// TwinCAT 3 PLC project PLC
// ProgramVersion: 3.1.4023.0
// libraries:
//   Tc2_Standard, * (Beckhoff Automation GmbH)
//   Tc2_System, * (Beckhoff Automation GmbH)
//   Tc3_Module, * (Beckhoff Automation GmbH)
// project tree:
//   / PlcTask.TcTTO
//   POUs/ MAIN.TcPOU
//   DUTs/IO/PdoEntries/ Status_B0753356.TcDUT, Status_05CE4FB5.TcDUT, Status_F2CE6D91.TcDUT, Status_AE4D73AB.TcDUT, Status_D1785240.TcDUT, Ctrl_AEDC374E.TcDUT, Status_36309700.TcDUT, Control_BD9A418F.TcDUT
//   DUTs/IO/PDOs/ InfoData_6F19DB2B.TcDUT, Channel_31CEFA7F.TcDUT, WcState_9091E0EB.TcDUT, Input_Type_NC_5EE69541.TcDUT, InfoData_32EB74EA.TcDUT, Channel_42CA91F7.TcDUT, WcState_0B2B16F9.TcDUT, AI_Standard_Channel_A8DF64E3.TcDUT, Ch_1_Al_Inputs_4794C083.TcDUT, InfoData_90184F0C.TcDUT, Ch_1_A1FAE759.TcDUT, AI_Standard_Channel_4A394481.TcDUT, AI_Standard_Channel_3D09D60D.TcDUT, RMB_Status_EE6B49B4.TcDUT, RMB_Value_INT_E9189C4B.TcDUT, RMB_Control_4997AEF6.TcDUT, AO_Output_Channel_BA7EBB7C.TcDUT, Ch_1_29D41289.TcDUT, ENC_Status_compact_BFB16BB4.TcDUT, ENC_Control_compact_2ED727EF.TcDUT, Status_Us_B1E819A2.TcDUT, Status_Up_B1E819A2.TcDUT, Status_Us_In_B1E819A2.TcDUT, Status_Us_Out_B1E819A2.TcDUT, Status_Uin_449D6AB5.TcDUT, Status_Uex_449D6AB5.TcDUT, Status_Uin_627CC56E.TcDUT, Status_Uex_834F3050.TcDUT, InfoData_E68C61CD.TcDUT, InfoData_2A97D6CF.TcDUT, Inputs_25A0042B.TcDUT, Outputs_2397A10E.TcDUT
//   DUTs/IO/Boxes/ EK1100_1FC0878B.TcDUT, EK1122_1FC0878B.TcDUT, ELX1052_6CC2DB6A.TcDUT, ELX1054_EF479B4E.TcDUT, ELX1058_7670813D.TcDUT, ELX2002_B0214940.TcDUT, ELX2008_E2806B95.TcDUT, ELX3152_AA20D87B.TcDUT, ELX3158_35AE5324.TcDUT, ELX3181_05065F7B.TcDUT, ELX3202_27F12237.TcDUT, ELX3204_B6248F5B.TcDUT, ELX3252_7FD1684B.TcDUT, ELX3312_BE98AB26.TcDUT, ELX3314_E65CDB1C.TcDUT, ELX3351_DF51302B.TcDUT, ELX4154_AB92710E.TcDUT, ELX4181_0949A6C0.TcDUT, ELX5151_C163EA3C.TcDUT, ELX9410_6BC01D14.TcDUT, ELX9410_089FA854.TcDUT, ELX9560_883C11A3.TcDUT, ELX9560_F22EDCF2.TcDUT
//   DUTs/IO/Devices/ SyncUnitTask_2D604ED5.TcDUT, SyncUnitTasks_6FEB8257.TcDUT, SyncUnits_99E584AF.TcDUT
//   DUTs/IO/Topology/ Beckhoff_ELXxxxxEK1122_3FD8C7C7.TcDUT, Beckhoff_ELXxxxx_62AA317A.TcDUT, EtherCAT_Master_ELXxxxx_D0B2812D.TcDUT
//   DUTs/IO/Base/ EtcSlaveBase_82538BE2.TcDUT, EtcSlaveBase_82538BE2.TcDUT, EtcSlaveBase_82538BE2.TcDUT, EtcSlaveTerminalBase_947E5A46.TcDUT, EtcSlaveBoxBase_77A0E4A7.TcDUT, EtcSlaveEndTerminalBase_866C7F0C.TcDUT, InputBase_8311D824.TcDUT, OutputBase_10CEE7DE.TcDUT, EtcMasterBase_62654B43.TcDUT
//   GVLs/ GVL_iXlinker.TcGVL
// real-time tasks:
//   TASK PlcTask: cycle T#10ms, priority 20, ADS port 350
// I/O:
//   DEVICE EtherCAT_Master_ELXxxxx, AmsNetId 172.20.30.238.11.1
//     Beckhoff ELXxxxx [EK1100 EtherCAT Coupler (2A E-Bus)]
//       Beckhoff ELXxxxxEK1122 [EK1122 2 port EtherCAT junction]
//         Beckhoff ELXxxxxsub EK1100 [EK1100 EtherCAT Coupler (2A E-Bus)]
//       A_0001(ELX1052-0000-0016) [ELX1052 2Ch. Dig. Input  NAMUR, Ex i]
//       A_0002(ELX1054-0000-0016) [ELX1054 4Ch. Dig. Input NAMUR, NO/NC, Ex i]
//       A_0003(ELX1058-0000-0016) [ELX1058 8Ch. Dig. Input NAMUR, NO/NC, Ex i]
//       A_0004(ELX2002-0000-0016) [ELX2002 2Ch. Dig. Output 24V, 45mA, Ex i]
//       A_0005(ELX2008-0000-0016) [ELX2008 8Ch. Dig. Output 24V, 30mA, Ex i]
//       A_0006(ELX3152-0000-0016) [ELX3152 2Ch. Ana. Input 0/4-20mA, Ex i]
//       A_0007(ELX3152-0000-0017) [ELX3152 2Ch. Ana. Input 0/4-20mA, Ex i]
//       A_0008(ELX3152-0090-0016) [ELX3152-0090 2Ch. Ana. Input 0/4-20mA, Ex i, TwinSAFE SC]
//       A_0009(ELX3152-0090-0017) [ELX3152-0090 2Ch. Ana. Input 0/4-20mA, Ex i, TwinSAFE SC]
//       A_0010(ELX3158-0000-0016) [ELX3158 8Ch. Ana. Input 4-20mA, Ex i]
//       A_0011(ELX3181-0000-0016) [ELX3181 1Ch. Ana. Input 4-20mA, HART, Ex i]
//         modules: Ch. 1, Ch. 1, Ch. 1, Ch. 1, Ch. 1, Ch. 1, Ch. 1, Ch. 1
//       A_0012(ELX3181-0000-0017) [ELX3181 1Ch. Ana. Input 4-20mA, HART, Ex i]
//         modules: Ch. 1, Ch. 1, Ch. 1, Ch. 1, Ch. 1, Ch. 1, Ch. 1, Ch. 1
//       A_0013(ELX3202-0000-0016) [ELX3202 2Ch. Ana. Input PT100 (RTD), Ex i]
//       A_0014(ELX3202-0090-0016) [ELX3202-0090 2Ch. Ana. Input PT100 (RTD), Ex i, TwinSAFE SC]
//       A_0015(ELX3204-0000-0016) [ELX3204 4Ch. Ana. Input PT100 (RTD), Ex i]
//       A_0016(ELX3204-0090-0016) [ELX3204-0090 4Ch. Ana. Input PT100 (RTD), Ex i, TwinSAFE SC]
//       A_0017(ELX3252-0000-0016) [ELX3252 2Ch. Ana. Input Potentiometer measurement, Ex i]
//       A_0018(ELX3312-0000-0016) [ELX3312 2Ch. Ana Input Thermocouple (TC), Ex i]
//       A_0019(ELX3312-0090-0016) [ELX3312-0090 2Ch. Ana Input Thermocouple (TC), Ex i, TwinSAFE SC]
//       A_0020(ELX3314-0000-0016) [ELX3314 4Ch. Ana Input Thermocouple (TC), Ex i]
//       A_0021(ELX3314-0090-0016) [ELX3314-0090 4Ch. Ana Input Thermocouple (TC), Ex i, TwinSAFE SC]
//       A_0022(ELX3351-0000-0016) [ELX3351 1-channel precise load cell analysis, Ex i]
//       A_0023(ELX3351-0090-0016) [ELX3351-0090 1-channel precise load cell analysis, TwinSAFE SC, Ex i]
//       A_0024(ELX4154-0000-0016) [ELX4154 4Ch. Ana. Output 4-20mA, 16 Bit, Ex i]
//       A_0025(ELX4181-0000-0016) [ELX4181 1-channel analog output terminal 0/4...20 mA, single-ended, HART, 16 bit, Ex i]
//         modules: Ch. 1
//       A_0026(ELX4181-0000-0017) [ELX4181 1-channel analog output terminal 0/4...20 mA, single-ended, HART, 16 bit, Ex i]
//         modules: Ch. 1
//       A_0027(ELX5151-0000-0016) [ELX5151 1Ch. Inc. Encoder NAMUR, Ex i]
//       A_0028(ELX5151-0090-0016) [ELX5151-0090 1Ch. Inc. Encoder NAMUR, Ex i, TwinSAFE SC]
//       A_0030(ELX9410-0000-0016) [ELX9410 E-Bus Power Supplier (Diagnostics)]
//       A_0031(ELX9410-0000-0017) [ELX9410 E-Bus Power Supplier (Diagnostics)]
//       A_0032(ELX9410-0000-0018) [ELX9410 E-Bus Power Supplier (Diagnostics)]
//       A_0033(ELX9560-0000-0016) [ELX9560 Power supply terminal 24V DC (350mA, isolated)]
//       A_0034(ELX9560-0000-0017) [ELX9560 Power supply terminal 24V DC (650mA, isolated)]
//       A_0035(ELX9560-0000-0018) [ELX9560 Power supply terminal 24V DC (650mA, isolated)]
// variable links:
//   PLC/PLC Instance <-> EtherCAT Master ELXxxxx/Beckhoff ELXxxxx
//     PlcTask Inputs/GVL_iXlinker.EtherCAT_Master_ELXxxxx.Beckhoff_ELXxxxx.InfoData.State <-> InfoData/State
//   PLC/PLC Instance <-> EtherCAT Master ELXxxxx/Beckhoff ELXxxxx/Beckhoff ELXxxxxEK1122
//     PlcTask Inputs/GVL_iXlinker.EtherCAT_Master_ELXxxxx.Beckhoff_ELXxxxx.Beckhoff_ELXxxxxEK1122.InfoData.State <-> InfoData/State
//   PLC/PLC Instance <-> EtherCAT Master ELXxxxx/Beckhoff ELXxxxx/Beckhoff ELXxxxxEK1122/Beckhoff ELXxxxxsub EK1100
//     PlcTask Inputs/GVL_iXlinker.EtherCAT_Master_ELXxxxx.Beckhoff_ELXxxxx.Beckhoff_ELXxxxxEK1122.Beckhoff_ELXxxxxsub_EK1100.InfoData.State <-> InfoData/State
//   PLC/PLC Instance <-> EtherCAT Master ELXxxxx/Beckhoff ELXxxxx/A_0001(ELX1052-0000-0016)
//     PlcTask Inputs/GVL_iXlinker.EtherCAT_Master_ELXxxxx.Beckhoff_ELXxxxx.A_0001_ELX1052_0000_0016.Channel_1.Input <-> Channel 1/Input
//     PlcTask Inputs/GVL_iXlinker.EtherCAT_Master_ELXxxxx.Beckhoff_ELXxxxx.A_0001_ELX1052_0000_0016.Channel_2.Input <-> Channel 2/Input
//     PlcTask Inputs/GVL_iXlinker.EtherCAT_Master_ELXxxxx.Beckhoff_ELXxxxx.A_0001_ELX1052_0000_0016.Channel_1.Error <-> Channel 1/Error
//     PlcTask Inputs/GVL_iXlinker.EtherCAT_Master_ELXxxxx.Beckhoff_ELXxxxx.A_0001_ELX1052_0000_0016.Channel_2.Error <-> Channel 2/Error
//     PlcTask Inputs/GVL_iXlinker.EtherCAT_Master_ELXxxxx.Beckhoff_ELXxxxx.A_0001_ELX1052_0000_0016.WcState.WcState <-> WcState/WcState
//     PlcTask Inputs/GVL_iXlinker.EtherCAT_Master_ELXxxxx.Beckhoff_ELXxxxx.A_0001_ELX1052_0000_0016.WcState.InputToggle <-> WcState/InputToggle
//     PlcTask Inputs/GVL_iXlinker.EtherCAT_Master_ELXxxxx.Beckhoff_ELXxxxx.A_0001_ELX1052_0000_0016.InfoData.State <-> InfoData/State
//   PLC/PLC Instance <-> EtherCAT Master ELXxxxx/Beckhoff ELXxxxx/A_0002(ELX1054-0000-0016)
//     PlcTask Inputs/GVL_iXlinker.EtherCAT_Master_ELXxxxx.Beckhoff_ELXxxxx.A_0002_ELX1054_0000_0016.Channel_1.Input <-> Channel 1/Input
//     PlcTask Inputs/GVL_iXlinker.EtherCAT_Master_ELXxxxx.Beckhoff_ELXxxxx.A_0002_ELX1054_0000_0016.Channel_2.Input <-> Channel 2/Input
//     PlcTask Inputs/GVL_iXlinker.EtherCAT_Master_ELXxxxx.Beckhoff_ELXxxxx.A_0002_ELX1054_0000_0016.Channel_3.Input <-> Channel 3/Input
//     PlcTask Inputs/GVL_iXlinker.EtherCAT_Master_ELXxxxx.Beckhoff_ELXxxxx.A_0002_ELX1054_0000_0016.Channel_4.Input <-> Channel 4/Input
//     PlcTask Inputs/GVL_iXlinker.EtherCAT_Master_ELXxxxx.Beckhoff_ELXxxxx.A_0002_ELX1054_0000_0016.Channel_1.Error <-> Channel 1/Error
//     PlcTask Inputs/GVL_iXlinker.EtherCAT_Master_ELXxxxx.Beckhoff_ELXxxxx.A_0002_ELX1054_0000_0016.Channel_2.Error <-> Channel 2/Error
//     PlcTask Inputs/GVL_iXlinker.EtherCAT_Master_ELXxxxx.Beckhoff_ELXxxxx.A_0002_ELX1054_0000_0016.Channel_3.Error <-> Channel 3/Error
//     PlcTask Inputs/GVL_iXlinker.EtherCAT_Master_ELXxxxx.Beckhoff_ELXxxxx.A_0002_ELX1054_0000_0016.Channel_4.Error <-> Channel 4/Error
//     PlcTask Inputs/GVL_iXlinker.EtherCAT_Master_ELXxxxx.Beckhoff_ELXxxxx.A_0002_ELX1054_0000_0016.Input_Type_NC.Channel[0] <-> Input Type NC/Channel 1
//     PlcTask Inputs/GVL_iXlinker.EtherCAT_Master_ELXxxxx.Beckhoff_ELXxxxx.A_0002_ELX1054_0000_0016.Input_Type_NC.Channel[1] <-> Input Type NC/Channel 2
//     PlcTask Inputs/GVL_iXlinker.EtherCAT_Master_ELXxxxx.Beckhoff_ELXxxxx.A_0002_ELX1054_0000_0016.Input_Type_NC.Channel[2] <-> Input Type NC/Channel 3
//     PlcTask Inputs/GVL_iXlinker.EtherCAT_Master_ELXxxxx.Beckhoff_ELXxxxx.A_0002_ELX1054_0000_0016.Input_Type_NC.Channel[3] <-> Input Type NC/Channel 4
//     PlcTask Inputs/GVL_iXlinker.EtherCAT_Master_ELXxxxx.Beckhoff_ELXxxxx.A_0002_ELX1054_0000_0016.WcState.WcState <-> WcState/WcState
//     PlcTask Inputs/GVL_iXlinker.EtherCAT_Master_ELXxxxx.Beckhoff_ELXxxxx.A_0002_ELX1054_0000_0016.WcState.InputToggle <-> WcState/InputToggle
//     PlcTask Inputs/GVL_iXlinker.EtherCAT_Master_ELXxxxx.Beckhoff_ELXxxxx.A_0002_ELX1054_0000_0016.InfoData.State <-> InfoData/State
//   PLC/PLC Instance <-> EtherCAT Master ELXxxxx/Beckhoff ELXxxxx/A_0003(ELX1058-0000-0016)
//     PlcTask Inputs/GVL_iXlinker.EtherCAT_Master_ELXxxxx.Beckhoff_ELXxxxx.A_0003_ELX1058_0000_0016.Channel_1.Input <-> Channel 1/Input
//     PlcTask Inputs/GVL_iXlinker.EtherCAT_Master_ELXxxxx.Beckhoff_ELXxxxx.A_0003_ELX1058_0000_0016.Channel_2.Input <-> Channel 2/Input
//     PlcTask Inputs/GVL_iXlinker.EtherCAT_Master_ELXxxxx.Beckhoff_ELXxxxx.A_0003_ELX1058_0000_0016.Channel_3.Input <-> Channel 3/Input
//     PlcTask Inputs/GVL_iXlinker.EtherCAT_Master_ELXxxxx.Beckhoff_ELXxxxx.A_0003_ELX1058_0000_0016.Channel_4.Input <-> Channel 4/Input
//     PlcTask Inputs/GVL_iXlinker.EtherCAT_Master_ELXxxxx.Beckhoff_ELXxxxx.A_0003_ELX1058_0000_0016.Channel_5.Input <-> Channel 5/Input
//     PlcTask Inputs/GVL_iXlinker.EtherCAT_Master_ELXxxxx.Beckhoff_ELXxxxx.A_0003_ELX1058_0000_0016.Channel_6.Input <-> Channel 6/Input
//     PlcTask Inputs/GVL_iXlinker.EtherCAT_Master_ELXxxxx.Beckhoff_ELXxxxx.A_0003_ELX1058_0000_0016.Channel_7.Input <-> Channel 7/Input
//     PlcTask Inputs/GVL_iXlinker.EtherCAT_Master_ELXxxxx.Beckhoff_ELXxxxx.A_0003_ELX1058_0000_0016.Channel_8.Input <-> Channel 8/Input
//     PlcTask Inputs/GVL_iXlinker.EtherCAT_Master_ELXxxxx.Beckhoff_ELXxxxx.A_0003_ELX1058_0000_0016.Channel_1.Error <-> Channel 1/Error
//     PlcTask Inputs/GVL_iXlinker.EtherCAT_Master_ELXxxxx.Beckhoff_ELXxxxx.A_0003_ELX1058_0000_0016.Channel_2.Error <-> Channel 2/Error
//     PlcTask Inputs/GVL_iXlinker.EtherCAT_Master_ELXxxxx.Beckhoff_ELXxxxx.A_0003_ELX1058_0000_0016.Channel_3.Error <-> Channel 3/Error
//     PlcTask Inputs/GVL_iXlinker.EtherCAT_Master_ELXxxxx.Beckhoff_ELXxxxx.A_0003_ELX1058_0000_0016.Channel_4.Error <-> Channel 4/Error
//     PlcTask Inputs/GVL_iXlinker.EtherCAT_Master_ELXxxxx.Beckhoff_ELXxxxx.A_0003_ELX1058_0000_0016.Channel_5.Error <-> Channel 5/Error
//     PlcTask Inputs/GVL_iXlinker.EtherCAT_Master_ELXxxxx.Beckhoff_ELXxxxx.A_0003_ELX1058_0000_0016.Channel_6.Error <-> Channel 6/Error
//     PlcTask Inputs/GVL_iXlinker.EtherCAT_Master_ELXxxxx.Beckhoff_ELXxxxx.A_0003_ELX1058_0000_0016.Channel_7.Error <-> Channel 7/Error
//     PlcTask Inputs/GVL_iXlinker.EtherCAT_Master_ELXxxxx.Beckhoff_ELXxxxx.A_0003_ELX1058_0000_0016.Channel_8.Error <-> Channel 8/Error
//     PlcTask Inputs/GVL_iXlinker.EtherCAT_Master_ELXxxxx.Beckhoff_ELXxxxx.A_0003_ELX1058_0000_0016.WcState.WcState <-> WcState/WcState
//     PlcTask Inputs/GVL_iXlinker.EtherCAT_Master_ELXxxxx.Beckhoff_ELXxxxx.A_0003_ELX1058_0000_0016.WcState.InputToggle <-> WcState/InputToggle
//     PlcTask Inputs/GVL_iXlinker.EtherCAT_Master_ELXxxxx.Beckhoff_ELXxxxx.A_0003_ELX1058_0000_0016.InfoData.AdsAddr <-> InfoData/AdsAddr
//     PlcTask Inputs/GVL_iXlinker.EtherCAT_Master_ELXxxxx.Beckhoff_ELXxxxx.A_0003_ELX1058_0000_0016.InfoData.State <-> InfoData/State
//   PLC/PLC Instance <-> EtherCAT Master ELXxxxx/Beckhoff ELXxxxx/A_0004(ELX2002-0000-0016)
//     PlcTask Outputs/GVL_iXlinker.EtherCAT_Master_ELXxxxx.Beckhoff_ELXxxxx.A_0004_ELX2002_0000_0016.Channel_1.Output <-> Channel 1/Output
//     PlcTask Outputs/GVL_iXlinker.EtherCAT_Master_ELXxxxx.Beckhoff_ELXxxxx.A_0004_ELX2002_0000_0016.Channel_2.Output <-> Channel 2/Output
//     PlcTask Inputs/GVL_iXlinker.EtherCAT_Master_ELXxxxx.Beckhoff_ELXxxxx.A_0004_ELX2002_0000_0016.WcState.WcState <-> WcState/WcState
//     PlcTask Inputs/GVL_iXlinker.EtherCAT_Master_ELXxxxx.Beckhoff_ELXxxxx.A_0004_ELX2002_0000_0016.InfoData.State <-> InfoData/State
//   PLC/PLC Instance <-> EtherCAT Master ELXxxxx/Beckhoff ELXxxxx/A_0005(ELX2008-0000-0016)
//     PlcTask Outputs/GVL_iXlinker.EtherCAT_Master_ELXxxxx.Beckhoff_ELXxxxx.A_0005_ELX2008_0000_0016.Channel_1.Output <-> Channel 1/Output
//     PlcTask Outputs/GVL_iXlinker.EtherCAT_Master_ELXxxxx.Beckhoff_ELXxxxx.A_0005_ELX2008_0000_0016.Channel_2.Output <-> Channel 2/Output
//     PlcTask Outputs/GVL_iXlinker.EtherCAT_Master_ELXxxxx.Beckhoff_ELXxxxx.A_0005_ELX2008_0000_0016.Channel_3.Output <-> Channel 3/Output
//     PlcTask Outputs/GVL_iXlinker.EtherCAT_Master_ELXxxxx.Beckhoff_ELXxxxx.A_0005_ELX2008_0000_0016.Channel_4.Output <-> Channel 4/Output
//     PlcTask Outputs/GVL_iXlinker.EtherCAT_Master_ELXxxxx.Beckhoff_ELXxxxx.A_0005_ELX2008_0000_0016.Channel_5.Output <-> Channel 5/Output
//     PlcTask Outputs/GVL_iXlinker.EtherCAT_Master_ELXxxxx.Beckhoff_ELXxxxx.A_0005_ELX2008_0000_0016.Channel_6.Output <-> Channel 6/Output
//     PlcTask Outputs/GVL_iXlinker.EtherCAT_Master_ELXxxxx.Beckhoff_ELXxxxx.A_0005_ELX2008_0000_0016.Channel_7.Output <-> Channel 7/Output
//     PlcTask Outputs/GVL_iXlinker.EtherCAT_Master_ELXxxxx.Beckhoff_ELXxxxx.A_0005_ELX2008_0000_0016.Channel_8.Output <-> Channel 8/Output
//     PlcTask Inputs/GVL_iXlinker.EtherCAT_Master_ELXxxxx.Beckhoff_ELXxxxx.A_0005_ELX2008_0000_0016.WcState.WcState <-> WcState/WcState
//     PlcTask Inputs/GVL_iXlinker.EtherCAT_Master_ELXxxxx.Beckhoff_ELXxxxx.A_0005_ELX2008_0000_0016.InfoData.State <-> InfoData/State
//   PLC/PLC Instance <-> EtherCAT Master ELXxxxx/Beckhoff ELXxxxx/A_0006(ELX3152-0000-0016)
//     PlcTask Inputs/GVL_iXlinker.EtherCAT_Master_ELXxxxx.Beckhoff_ELXxxxx.A_0006_ELX3152_0000_0016.AI_Standard_Channel_1.Status/Underrange <-> AI Standard Channel 1/Status/Underrange
//     PlcTask Inputs/GVL_iXlinker.EtherCAT_Master_ELXxxxx.Beckhoff_ELXxxxx.A_0006_ELX3152_0000_0016.AI_Standard_Channel_2.Status/Underrange <-> AI Standard Channel 2/Status/Underrange
//     PlcTask Inputs/GVL_iXlinker.EtherCAT_Master_ELXxxxx.Beckhoff_ELXxxxx.A_0006_ELX3152_0000_0016.AI_Standard_Channel_1.Status/Overrange <-> AI Standard Channel 1/Status/Overrange
//     PlcTask Inputs/GVL_iXlinker.EtherCAT_Master_ELXxxxx.Beckhoff_ELXxxxx.A_0006_ELX3152_0000_0016.AI_Standard_Channel_2.Status/Overrange <-> AI Standard Channel 2/Status/Overrange
//     PlcTask Inputs/GVL_iXlinker.EtherCAT_Master_ELXxxxx.Beckhoff_ELXxxxx.A_0006_ELX3152_0000_0016.AI_Standard_Channel_1.Status/Limit_1 <-> AI Standard Channel 1/Status/Limit 1
//     PlcTask Inputs/GVL_iXlinker.EtherCAT_Master_ELXxxxx.Beckhoff_ELXxxxx.A_0006_ELX3152_0000_0016.AI_Standard_Channel_1.Status/Limit_2 <-> AI Standard Channel 1/Status/Limit 2
//     PlcTask Inputs/GVL_iXlinker.EtherCAT_Master_ELXxxxx.Beckhoff_ELXxxxx.A_0006_ELX3152_0000_0016.AI_Standard_Channel_2.Status/Limit_1 <-> AI Standard Channel 2/Status/Limit 1
//     PlcTask Inputs/GVL_iXlinker.EtherCAT_Master_ELXxxxx.Beckhoff_ELXxxxx.A_0006_ELX3152_0000_0016.AI_Standard_Channel_2.Status/Limit_2 <-> AI Standard Channel 2/Status/Limit 2
//     PlcTask Inputs/GVL_iXlinker.EtherCAT_Master_ELXxxxx.Beckhoff_ELXxxxx.A_0006_ELX3152_0000_0016.AI_Standard_Channel_1.Status/Error <-> AI Standard Channel 1/Status/Error
//     PlcTask Inputs/GVL_iXlinker.EtherCAT_Master_ELXxxxx.Beckhoff_ELXxxxx.A_0006_ELX3152_0000_0016.AI_Standard_Channel_2.Status/Error <-> AI Standard Channel 2/Status/Error
//     PlcTask Inputs/GVL_iXlinker.EtherCAT_Master_ELXxxxx.Beckhoff_ELXxxxx.A_0006_ELX3152_0000_0016.AI_Standard_Channel_1.Status/Sync_error <-> AI Standard Channel 1/Status/Sync error
//     PlcTask Inputs/GVL_iXlinker.EtherCAT_Master_ELXxxxx.Beckhoff_ELXxxxx.A_0006_ELX3152_0000_0016.AI_Standard_Channel_2.Status/Sync_error <-> AI Standard Channel 2/Status/Sync error
//     PlcTask Inputs/GVL_iXlinker.EtherCAT_Master_ELXxxxx.Beckhoff_ELXxxxx.A_0006_ELX3152_0000_0016.AI_Standard_Channel_1.Status/TxPDO_State <-> AI Standard Channel 1/Status/TxPDO State
//     PlcTask Inputs/GVL_iXlinker.EtherCAT_Master_ELXxxxx.Beckhoff_ELXxxxx.A_0006_ELX3152_0000_0016.AI_Standard_Channel_2.Status/TxPDO_State <-> AI Standard Channel 2/Status/TxPDO State
//     PlcTask Inputs/GVL_iXlinker.EtherCAT_Master_ELXxxxx.Beckhoff_ELXxxxx.A_0006_ELX3152_0000_0016.AI_Standard_Channel_1.Status/TxPDO_Toggle <-> AI Standard Channel 1/Status/TxPDO Toggle
//     PlcTask Inputs/GVL_iXlinker.EtherCAT_Master_ELXxxxx.Beckhoff_ELXxxxx.A_0006_ELX3152_0000_0016.AI_Standard_Channel_2.Status/TxPDO_Toggle <-> AI Standard Channel 2/Status/TxPDO Toggle
//     PlcTask Inputs/GVL_iXlinker.EtherCAT_Master_ELXxxxx.Beckhoff_ELXxxxx.A_0006_ELX3152_0000_0016.AI_Standard_Channel_1.Value <-> AI Standard Channel 1/Value
//     PlcTask Inputs/GVL_iXlinker.EtherCAT_Master_ELXxxxx.Beckhoff_ELXxxxx.A_0006_ELX3152_0000_0016.AI_Standard_Channel_2.Value <-> AI Standard Channel 2/Value
//     PlcTask Inputs/GVL_iXlinker.EtherCAT_Master_ELXxxxx.Beckhoff_ELXxxxx.A_0006_ELX3152_0000_0016.WcState.WcState <-> WcState/WcState
//     PlcTask Inputs/GVL_iXlinker.EtherCAT_Master_ELXxxxx.Beckhoff_ELXxxxx.A_0006_ELX3152_0000_0016.WcState.InputToggle <-> WcState/InputToggle
//     PlcTask Inputs/GVL_iXlinker.EtherCAT_Master_ELXxxxx.Beckhoff_ELXxxxx.A_0006_ELX3152_0000_0016.InfoData.AdsAddr <-> InfoData/AdsAddr
//     PlcTask Inputs/GVL_iXlinker.EtherCAT_Master_ELXxxxx.Beckhoff_ELXxxxx.A_0006_ELX3152_0000_0016.InfoData.State <-> InfoData/State
//   PLC/PLC Instance <-> EtherCAT Master ELXxxxx/Beckhoff ELXxxxx/A_0007(ELX3152-0000-0017)
//     PlcTask Inputs/GVL_iXlinker.EtherCAT_Master_ELXxxxx.Beckhoff_ELXxxxx.A_0007_ELX3152_0000_0017.AI_Standard_Channel_1.Status/Underrange <-> AI Standard Channel 1/Status/Underrange
//     PlcTask Inputs/GVL_iXlinker.EtherCAT_Master_ELXxxxx.Beckhoff_ELXxxxx.A_0007_ELX3152_0000_0017.AI_Standard_Channel_2.Status/Underrange <-> AI Standard Channel 2/Status/Underrange
//     PlcTask Inputs/GVL_iXlinker.EtherCAT_Master_ELXxxxx.Beckhoff_ELXxxxx.A_0007_ELX3152_0000_0017.AI_Standard_Channel_1.Status/Overrange <-> AI Standard Channel 1/Status/Overrange
//     PlcTask Inputs/GVL_iXlinker.EtherCAT_Master_ELXxxxx.Beckhoff_ELXxxxx.A_0007_ELX3152_0000_0017.AI_Standard_Channel_2.Status/Overrange <-> AI Standard Channel 2/Status/Overrange
//     PlcTask Inputs/GVL_iXlinker.EtherCAT_Master_ELXxxxx.Beckhoff_ELXxxxx.A_0007_ELX3152_0000_0017.AI_Standard_Channel_1.Status/Limit_1 <-> AI Standard Channel 1/Status/Limit 1
//     PlcTask Inputs/GVL_iXlinker.EtherCAT_Master_ELXxxxx.Beckhoff_ELXxxxx.A_0007_ELX3152_0000_0017.AI_Standard_Channel_1.Status/Limit_2 <-> AI Standard Channel 1/Status/Limit 2
//     PlcTask Inputs/GVL_iXlinker.EtherCAT_Master_ELXxxxx.Beckhoff_ELXxxxx.A_0007_ELX3152_0000_0017.AI_Standard_Channel_2.Status/Limit_1 <-> AI Standard Channel 2/Status/Limit 1
//     PlcTask Inputs/GVL_iXlinker.EtherCAT_Master_ELXxxxx.Beckhoff_ELXxxxx.A_0007_ELX3152_0000_0017.AI_Standard_Channel_2.Status/Limit_2 <-> AI Standard Channel 2/Status/Limit 2
//     PlcTask Inputs/GVL_iXlinker.EtherCAT_Master_ELXxxxx.Beckhoff_ELXxxxx.A_0007_ELX3152_0000_0017.AI_Standard_Channel_1.Status/Error <-> AI Standard Channel 1/Status/Error
//     PlcTask Inputs/GVL_iXlinker.EtherCAT_Master_ELXxxxx.Beckhoff_ELXxxxx.A_0007_ELX3152_0000_0017.AI_Standard_Channel_2.Status/Error <-> AI Standard Channel 2/Status/Error
//     PlcTask Inputs/GVL_iXlinker.EtherCAT_Master_ELXxxxx.Beckhoff_ELXxxxx.A_0007_ELX3152_0000_0017.AI_Standard_Channel_1.Status/Sync_error <-> AI Standard Channel 1/Status/Sync error
//     PlcTask Inputs/GVL_iXlinker.EtherCAT_Master_ELXxxxx.Beckhoff_ELXxxxx.A_0007_ELX3152_0000_0017.AI_Standard_Channel_2.Status/Sync_error <-> AI Standard Channel 2/Status/Sync error
//     PlcTask Inputs/GVL_iXlinker.EtherCAT_Master_ELXxxxx.Beckhoff_ELXxxxx.A_0007_ELX3152_0000_0017.AI_Standard_Channel_1.Status/TxPDO_State <-> AI Standard Channel 1/Status/TxPDO State
//     PlcTask Inputs/GVL_iXlinker.EtherCAT_Master_ELXxxxx.Beckhoff_ELXxxxx.A_0007_ELX3152_0000_0017.AI_Standard_Channel_2.Status/TxPDO_State <-> AI Standard Channel 2/Status/TxPDO State
//     PlcTask Inputs/GVL_iXlinker.EtherCAT_Master_ELXxxxx.Beckhoff_ELXxxxx.A_0007_ELX3152_0000_0017.AI_Standard_Channel_1.Status/TxPDO_Toggle <-> AI Standard Channel 1/Status/TxPDO Toggle
//     PlcTask Inputs/GVL_iXlinker.EtherCAT_Master_ELXxxxx.Beckhoff_ELXxxxx.A_0007_ELX3152_0000_0017.AI_Standard_Channel_2.Status/TxPDO_Toggle <-> AI Standard Channel 2/Status/TxPDO Toggle
//     PlcTask Inputs/GVL_iXlinker.EtherCAT_Master_ELXxxxx.Beckhoff_ELXxxxx.A_0007_ELX3152_0000_0017.AI_Standard_Channel_1.Value <-> AI Standard Channel 1/Value
//     PlcTask Inputs/GVL_iXlinker.EtherCAT_Master_ELXxxxx.Beckhoff_ELXxxxx.A_0007_ELX3152_0000_0017.AI_Standard_Channel_2.Value <-> AI Standard Channel 2/Value
//     PlcTask Inputs/GVL_iXlinker.EtherCAT_Master_ELXxxxx.Beckhoff_ELXxxxx.A_0007_ELX3152_0000_0017.WcState.WcState <-> WcState/WcState
//     PlcTask Inputs/GVL_iXlinker.EtherCAT_Master_ELXxxxx.Beckhoff_ELXxxxx.A_0007_ELX3152_0000_0017.WcState.InputToggle <-> WcState/InputToggle
//     PlcTask Inputs/GVL_iXlinker.EtherCAT_Master_ELXxxxx.Beckhoff_ELXxxxx.A_0007_ELX3152_0000_0017.InfoData.AdsAddr <-> InfoData/AdsAddr
//     PlcTask Inputs/GVL_iXlinker.EtherCAT_Master_ELXxxxx.Beckhoff_ELXxxxx.A_0007_ELX3152_0000_0017.InfoData.State <-> InfoData/State
//   PLC/PLC Instance <-> EtherCAT Master ELXxxxx/Beckhoff ELXxxxx/A_0008(ELX3152-0090-0016)
//     PlcTask Inputs/GVL_iXlinker.EtherCAT_Master_ELXxxxx.Beckhoff_ELXxxxx.A_0008_ELX3152_0090_0016.AI_Standard_Channel_1.Status/Underrange <-> AI Standard Channel 1/Status/Underrange
//     PlcTask Inputs/GVL_iXlinker.EtherCAT_Master_ELXxxxx.Beckhoff_ELXxxxx.A_0008_ELX3152_0090_0016.AI_Standard_Channel_2.Status/Underrange <-> AI Standard Channel 2/Status/Underrange
//     PlcTask Inputs/GVL_iXlinker.EtherCAT_Master_ELXxxxx.Beckhoff_ELXxxxx.A_0008_ELX3152_0090_0016.AI_Standard_Channel_1.Status/Overrange <-> AI Standard Channel 1/Status/Overrange
//     PlcTask Inputs/GVL_iXlinker.EtherCAT_Master_ELXxxxx.Beckhoff_ELXxxxx.A_0008_ELX3152_0090_0016.AI_Standard_Channel_2.Status/Overrange <-> AI Standard Channel 2/Status/Overrange
//     PlcTask Inputs/GVL_iXlinker.EtherCAT_Master_ELXxxxx.Beckhoff_ELXxxxx.A_0008_ELX3152_0090_0016.AI_Standard_Channel_1.Status/Limit_1 <-> AI Standard Channel 1/Status/Limit 1
//     PlcTask Inputs/GVL_iXlinker.EtherCAT_Master_ELXxxxx.Beckhoff_ELXxxxx.A_0008_ELX3152_0090_0016.AI_Standard_Channel_1.Status/Limit_2 <-> AI Standard Channel 1/Status/Limit 2
//     PlcTask Inputs/GVL_iXlinker.EtherCAT_Master_ELXxxxx.Beckhoff_ELXxxxx.A_0008_ELX3152_0090_0016.AI_Standard_Channel_2.Status/Limit_1 <-> AI Standard Channel 2/Status/Limit 1
//     PlcTask Inputs/GVL_iXlinker.EtherCAT_Master_ELXxxxx.Beckhoff_ELXxxxx.A_0008_ELX3152_0090_0016.AI_Standard_Channel_2.Status/Limit_2 <-> AI Standard Channel 2/Status/Limit 2
//     PlcTask Inputs/GVL_iXlinker.EtherCAT_Master_ELXxxxx.Beckhoff_ELXxxxx.A_0008_ELX3152_0090_0016.AI_Standard_Channel_1.Status/Error <-> AI Standard Channel 1/Status/Error
//     PlcTask Inputs/GVL_iXlinker.EtherCAT_Master_ELXxxxx.Beckhoff_ELXxxxx.A_0008_ELX3152_0090_0016.AI_Standard_Channel_2.Status/Error <-> AI Standard Channel 2/Status/Error
//     PlcTask Inputs/GVL_iXlinker.EtherCAT_Master_ELXxxxx.Beckhoff_ELXxxxx.A_0008_ELX3152_0090_0016.AI_Standard_Channel_1.Status/Sync_error <-> AI Standard Channel 1/Status/Sync error
//     PlcTask Inputs/GVL_iXlinker.EtherCAT_Master_ELXxxxx.Beckhoff_ELXxxxx.A_0008_ELX3152_0090_0016.AI_Standard_Channel_2.Status/Sync_error <-> AI Standard Channel 2/Status/Sync error
//     PlcTask Inputs/GVL_iXlinker.EtherCAT_Master_ELXxxxx.Beckhoff_ELXxxxx.A_0008_ELX3152_0090_0016.AI_Standard_Channel_1.Status/TxPDO_State <-> AI Standard Channel 1/Status/TxPDO State
//     PlcTask Inputs/GVL_iXlinker.EtherCAT_Master_ELXxxxx.Beckhoff_ELXxxxx.A_0008_ELX3152_0090_0016.AI_Standard_Channel_2.Status/TxPDO_State <-> AI Standard Channel 2/Status/TxPDO State
//     PlcTask Inputs/GVL_iXlinker.EtherCAT_Master_ELXxxxx.Beckhoff_ELXxxxx.A_0008_ELX3152_0090_0016.AI_Standard_Channel_1.Status/TxPDO_Toggle <-> AI Standard Channel 1/Status/TxPDO Toggle
//     PlcTask Inputs/GVL_iXlinker.EtherCAT_Master_ELXxxxx.Beckhoff_ELXxxxx.A_0008_ELX3152_0090_0016.AI_Standard_Channel_2.Status/TxPDO_Toggle <-> AI Standard Channel 2/Status/TxPDO Toggle
//     PlcTask Inputs/GVL_iXlinker.EtherCAT_Master_ELXxxxx.Beckhoff_ELXxxxx.A_0008_ELX3152_0090_0016.AI_Standard_Channel_1.Value <-> AI Standard Channel 1/Value
//     PlcTask Inputs/GVL_iXlinker.EtherCAT_Master_ELXxxxx.Beckhoff_ELXxxxx.A_0008_ELX3152_0090_0016.AI_Standard_Channel_2.Value <-> AI Standard Channel 2/Value
//     PlcTask Inputs/GVL_iXlinker.EtherCAT_Master_ELXxxxx.Beckhoff_ELXxxxx.A_0008_ELX3152_0090_0016.WcState.WcState <-> WcState/WcState
//     PlcTask Inputs/GVL_iXlinker.EtherCAT_Master_ELXxxxx.Beckhoff_ELXxxxx.A_0008_ELX3152_0090_0016.WcState.InputToggle <-> WcState/InputToggle
//     PlcTask Inputs/GVL_iXlinker.EtherCAT_Master_ELXxxxx.Beckhoff_ELXxxxx.A_0008_ELX3152_0090_0016.InfoData.AdsAddr <-> InfoData/AdsAddr
//     PlcTask Inputs/GVL_iXlinker.EtherCAT_Master_ELXxxxx.Beckhoff_ELXxxxx.A_0008_ELX3152_0090_0016.InfoData.State <-> InfoData/State
//   PLC/PLC Instance <-> EtherCAT Master ELXxxxx/Beckhoff ELXxxxx/A_0009(ELX3152-0090-0017)
//     PlcTask Inputs/GVL_iXlinker.EtherCAT_Master_ELXxxxx.Beckhoff_ELXxxxx.A_0009_ELX3152_0090_0017.AI_Standard_Channel_1.Status/Underrange <-> AI Standard Channel 1/Status/Underrange
//     PlcTask Inputs/GVL_iXlinker.EtherCAT_Master_ELXxxxx.Beckhoff_ELXxxxx.A_0009_ELX3152_0090_0017.AI_Standard_Channel_2.Status/Underrange <-> AI Standard Channel 2/Status/Underrange
//     PlcTask Inputs/GVL_iXlinker.EtherCAT_Master_ELXxxxx.Beckhoff_ELXxxxx.A_0009_ELX3152_0090_0017.AI_Standard_Channel_1.Status/Overrange <-> AI Standard Channel 1/Status/Overrange
//     PlcTask Inputs/GVL_iXlinker.EtherCAT_Master_ELXxxxx.Beckhoff_ELXxxxx.A_0009_ELX3152_0090_0017.AI_Standard_Channel_2.Status/Overrange <-> AI Standard Channel 2/Status/Overrange
//     PlcTask Inputs/GVL_iXlinker.EtherCAT_Master_ELXxxxx.Beckhoff_ELXxxxx.A_0009_ELX3152_0090_0017.AI_Standard_Channel_1.Status/Limit_1 <-> AI Standard Channel 1/Status/Limit 1
//     PlcTask Inputs/GVL_iXlinker.EtherCAT_Master_ELXxxxx.Beckhoff_ELXxxxx.A_0009_ELX3152_0090_0017.AI_Standard_Channel_1.Status/Limit_2 <-> AI Standard Channel 1/Status/Limit 2
//     PlcTask Inputs/GVL_iXlinker.EtherCAT_Master_ELXxxxx.Beckhoff_ELXxxxx.A_0009_ELX3152_0090_0017.AI_Standard_Channel_2.Status/Limit_1 <-> AI Standard Channel 2/Status/Limit 1
//     PlcTask Inputs/GVL_iXlinker.EtherCAT_Master_ELXxxxx.Beckhoff_ELXxxxx.A_0009_ELX3152_0090_0017.AI_Standard_Channel_2.Status/Limit_2 <-> AI Standard Channel 2/Status/Limit 2
//     PlcTask Inputs/GVL_iXlinker.EtherCAT_Master_ELXxxxx.Beckhoff_ELXxxxx.A_0009_ELX3152_0090_0017.AI_Standard_Channel_1.Status/Error <-> AI Standard Channel 1/Status/Error
//     PlcTask Inputs/GVL_iXlinker.EtherCAT_Master_ELXxxxx.Beckhoff_ELXxxxx.A_0009_ELX3152_0090_0017.AI_Standard_Channel_2.Status/Error <-> AI Standard Channel 2/Status/Error
//     PlcTask Inputs/GVL_iXlinker.EtherCAT_Master_ELXxxxx.Beckhoff_ELXxxxx.A_0009_ELX3152_0090_0017.AI_Standard_Channel_1.Status/Sync_error <-> AI Standard Channel 1/Status/Sync error
//     PlcTask Inputs/GVL_iXlinker.EtherCAT_Master_ELXxxxx.Beckhoff_ELXxxxx.A_0009_ELX3152_0090_0017.AI_Standard_Channel_2.Status/Sync_error <-> AI Standard Channel 2/Status/Sync error
//     PlcTask Inputs/GVL_iXlinker.EtherCAT_Master_ELXxxxx.Beckhoff_ELXxxxx.A_0009_ELX3152_0090_0017.AI_Standard_Channel_1.Status/TxPDO_State <-> AI Standard Channel 1/Status/TxPDO State
//     PlcTask Inputs/GVL_iXlinker.EtherCAT_Master_ELXxxxx.Beckhoff_ELXxxxx.A_0009_ELX3152_0090_0017.AI_Standard_Channel_2.Status/TxPDO_State <-> AI Standard Channel 2/Status/TxPDO State
//     PlcTask Inputs/GVL_iXlinker.EtherCAT_Master_ELXxxxx.Beckhoff_ELXxxxx.A_0009_ELX3152_0090_0017.AI_Standard_Channel_1.Status/TxPDO_Toggle <-> AI Standard Channel 1/Status/TxPDO Toggle
//     PlcTask Inputs/GVL_iXlinker.EtherCAT_Master_ELXxxxx.Beckhoff_ELXxxxx.A_0009_ELX3152_0090_0017.AI_Standard_Channel_2.Status/TxPDO_Toggle <-> AI Standard Channel 2/Status/TxPDO Toggle
//     PlcTask Inputs/GVL_iXlinker.EtherCAT_Master_ELXxxxx.Beckhoff_ELXxxxx.A_0009_ELX3152_0090_0017.AI_Standard_Channel_1.Value <-> AI Standard Channel 1/Value
//     PlcTask Inputs/GVL_iXlinker.EtherCAT_Master_ELXxxxx.Beckhoff_ELXxxxx.A_0009_ELX3152_0090_0017.AI_Standard_Channel_2.Value <-> AI Standard Channel 2/Value
//     PlcTask Inputs/GVL_iXlinker.EtherCAT_Master_ELXxxxx.Beckhoff_ELXxxxx.A_0009_ELX3152_0090_0017.WcState.WcState <-> WcState/WcState
//     PlcTask Inputs/GVL_iXlinker.EtherCAT_Master_ELXxxxx.Beckhoff_ELXxxxx.A_0009_ELX3152_0090_0017.WcState.InputToggle <-> WcState/InputToggle
//     PlcTask Inputs/GVL_iXlinker.EtherCAT_Master_ELXxxxx.Beckhoff_ELXxxxx.A_0009_ELX3152_0090_0017.InfoData.AdsAddr <-> InfoData/AdsAddr
//     PlcTask Inputs/GVL_iXlinker.EtherCAT_Master_ELXxxxx.Beckhoff_ELXxxxx.A_0009_ELX3152_0090_0017.InfoData.State <-> InfoData/State
//   PLC/PLC Instance <-> EtherCAT Master ELXxxxx/Beckhoff ELXxxxx/A_0010(ELX3158-0000-0016)
//     PlcTask Inputs/GVL_iXlinker.EtherCAT_Master_ELXxxxx.Beckhoff_ELXxxxx.A_0010_ELX3158_0000_0016.AI_Standard_Channel_1.Status/Underrange <-> AI Standard Channel 1/Status/Underrange
//     PlcTask Inputs/GVL_iXlinker.EtherCAT_Master_ELXxxxx.Beckhoff_ELXxxxx.A_0010_ELX3158_0000_0016.AI_Standard_Channel_2.Status/Underrange <-> AI Standard Channel 2/Status/Underrange
//     PlcTask Inputs/GVL_iXlinker.EtherCAT_Master_ELXxxxx.Beckhoff_ELXxxxx.A_0010_ELX3158_0000_0016.AI_Standard_Channel_3.Status/Underrange <-> AI Standard Channel 3/Status/Underrange
//     PlcTask Inputs/GVL_iXlinker.EtherCAT_Master_ELXxxxx.Beckhoff_ELXxxxx.A_0010_ELX3158_0000_0016.AI_Standard_Channel_4.Status/Underrange <-> AI Standard Channel 4/Status/Underrange
//     PlcTask Inputs/GVL_iXlinker.EtherCAT_Master_ELXxxxx.Beckhoff_ELXxxxx.A_0010_ELX3158_0000_0016.AI_Standard_Channel_5.Status/Underrange <-> AI Standard Channel 5/Status/Underrange
//     PlcTask Inputs/GVL_iXlinker.EtherCAT_Master_ELXxxxx.Beckhoff_ELXxxxx.A_0010_ELX3158_0000_0016.AI_Standard_Channel_6.Status/Underrange <-> AI Standard Channel 6/Status/Underrange
//     PlcTask Inputs/GVL_iXlinker.EtherCAT_Master_ELXxxxx.Beckhoff_ELXxxxx.A_0010_ELX3158_0000_0016.AI_Standard_Channel_7.Status/Underrange <-> AI Standard Channel 7/Status/Underrange
//     PlcTask Inputs/GVL_iXlinker.EtherCAT_Master_ELXxxxx.Beckhoff_ELXxxxx.A_0010_ELX3158_0000_0016.AI_Standard_Channel_8.Status/Underrange <-> AI Standard Channel 8/Status/Underrange
//     PlcTask Inputs/GVL_iXlinker.EtherCAT_Master_ELXxxxx.Beckhoff_ELXxxxx.A_0010_ELX3158_0000_0016.AI_Standard_Channel_1.Status/Overrange <-> AI Standard Channel 1/Status/Overrange
//     PlcTask Inputs/GVL_iXlinker.EtherCAT_Master_ELXxxxx.Beckhoff_ELXxxxx.A_0010_ELX3158_0000_0016.AI_Standard_Channel_2.Status/Overrange <-> AI Standard Channel 2/Status/Overrange
//     PlcTask Inputs/GVL_iXlinker.EtherCAT_Master_ELXxxxx.Beckhoff_ELXxxxx.A_0010_ELX3158_0000_0016.AI_Standard_Channel_3.Status/Overrange <-> AI Standard Channel 3/Status/Overrange
//     PlcTask Inputs/GVL_iXlinker.EtherCAT_Master_ELXxxxx.Beckhoff_ELXxxxx.A_0010_ELX3158_0000_0016.AI_Standard_Channel_4.Status/Overrange <-> AI Standard Channel 4/Status/Overrange
//     PlcTask Inputs/GVL_iXlinker.EtherCAT_Master_ELXxxxx.Beckhoff_ELXxxxx.A_0010_ELX3158_0000_0016.AI_Standard_Channel_5.Status/Overrange <-> AI Standard Channel 5/Status/Overrange
//     PlcTask Inputs/GVL_iXlinker.EtherCAT_Master_ELXxxxx.Beckhoff_ELXxxxx.A_0010_ELX3158_0000_0016.AI_Standard_Channel_6.Status/Overrange <-> AI Standard Channel 6/Status/Overrange
//     PlcTask Inputs/GVL_iXlinker.EtherCAT_Master_ELXxxxx.Beckhoff_ELXxxxx.A_0010_ELX3158_0000_0016.AI_Standard_Channel_7.Status/Overrange <-> AI Standard Channel 7/Status/Overrange
//     PlcTask Inputs/GVL_iXlinker.EtherCAT_Master_ELXxxxx.Beckhoff_ELXxxxx.A_0010_ELX3158_0000_0016.AI_Standard_Channel_8.Status/Overrange <-> AI Standard Channel 8/Status/Overrange
//     PlcTask Inputs/GVL_iXlinker.EtherCAT_Master_ELXxxxx.Beckhoff_ELXxxxx.A_0010_ELX3158_0000_0016.AI_Standard_Channel_1.Status/Limit_1 <-> AI Standard Channel 1/Status/Limit 1
//     PlcTask Inputs/GVL_iXlinker.EtherCAT_Master_ELXxxxx.Beckhoff_ELXxxxx.A_0010_ELX3158_0000_0016.AI_Standard_Channel_1.Status/Limit_2 <-> AI Standard Channel 1/Status/Limit 2
//     PlcTask Inputs/GVL_iXlinker.EtherCAT_Master_ELXxxxx.Beckhoff_ELXxxxx.A_0010_ELX3158_0000_0016.AI_Standard_Channel_2.Status/Limit_1 <-> AI Standard Channel 2/Status/Limit 1
//     PlcTask Inputs/GVL_iXlinker.EtherCAT_Master_ELXxxxx.Beckhoff_ELXxxxx.A_0010_ELX3158_0000_0016.AI_Standard_Channel_2.Status/Limit_2 <-> AI Standard Channel 2/Status/Limit 2
//     PlcTask Inputs/GVL_iXlinker.EtherCAT_Master_ELXxxxx.Beckhoff_ELXxxxx.A_0010_ELX3158_0000_0016.AI_Standard_Channel_3.Status/Limit_1 <-> AI Standard Channel 3/Status/Limit 1
//     PlcTask Inputs/GVL_iXlinker.EtherCAT_Master_ELXxxxx.Beckhoff_ELXxxxx.A_0010_ELX3158_0000_0016.AI_Standard_Channel_3.Status/Limit_2 <-> AI Standard Channel 3/Status/Limit 2
//     PlcTask Inputs/GVL_iXlinker.EtherCAT_Master_ELXxxxx.Beckhoff_ELXxxxx.A_0010_ELX3158_0000_0016.AI_Standard_Channel_4.Status/Limit_1 <-> AI Standard Channel 4/Status/Limit 1
//     PlcTask Inputs/GVL_iXlinker.EtherCAT_Master_ELXxxxx.Beckhoff_ELXxxxx.A_0010_ELX3158_0000_0016.AI_Standard_Channel_4.Status/Limit_2 <-> AI Standard Channel 4/Status/Limit 2
//     PlcTask Inputs/GVL_iXlinker.EtherCAT_Master_ELXxxxx.Beckhoff_ELXxxxx.A_0010_ELX3158_0000_0016.AI_Standard_Channel_5.Status/Limit_1 <-> AI Standard Channel 5/Status/Limit 1
//     PlcTask Inputs/GVL_iXlinker.EtherCAT_Master_ELXxxxx.Beckhoff_ELXxxxx.A_0010_ELX3158_0000_0016.AI_Standard_Channel_5.Status/Limit_2 <-> AI Standard Channel 5/Status/Limit 2
//     PlcTask Inputs/GVL_iXlinker.EtherCAT_Master_ELXxxxx.Beckhoff_ELXxxxx.A_0010_ELX3158_0000_0016.AI_Standard_Channel_6.Status/Limit_1 <-> AI Standard Channel 6/Status/Limit 1
//     PlcTask Inputs/GVL_iXlinker.EtherCAT_Master_ELXxxxx.Beckhoff_ELXxxxx.A_0010_ELX3158_0000_0016.AI_Standard_Channel_6.Status/Limit_2 <-> AI Standard Channel 6/Status/Limit 2
//     PlcTask Inputs/GVL_iXlinker.EtherCAT_Master_ELXxxxx.Beckhoff_ELXxxxx.A_0010_ELX3158_0000_0016.AI_Standard_Channel_7.Status/Limit_1 <-> AI Standard Channel 7/Status/Limit 1
//     PlcTask Inputs/GVL_iXlinker.EtherCAT_Master_ELXxxxx.Beckhoff_ELXxxxx.A_0010_ELX3158_0000_0016.AI_Standard_Channel_7.Status/Limit_2 <-> AI Standard Channel 7/Status/Limit 2
//     PlcTask Inputs/GVL_iXlinker.EtherCAT_Master_ELXxxxx.Beckhoff_ELXxxxx.A_0010_ELX3158_0000_0016.AI_Standard_Channel_8.Status/Limit_1 <-> AI Standard Channel 8/Status/Limit 1
//     PlcTask Inputs/GVL_iXlinker.EtherCAT_Master_ELXxxxx.Beckhoff_ELXxxxx.A_0010_ELX3158_0000_0016.AI_Standard_Channel_8.Status/Limit_2 <-> AI Standard Channel 8/Status/Limit 2
//     PlcTask Inputs/GVL_iXlinker.EtherCAT_Master_ELXxxxx.Beckhoff_ELXxxxx.A_0010_ELX3158_0000_0016.AI_Standard_Channel_1.Status/Error <-> AI Standard Channel 1/Status/Error
//     PlcTask Inputs/GVL_iXlinker.EtherCAT_Master_ELXxxxx.Beckhoff_ELXxxxx.A_0010_ELX3158_0000_0016.AI_Standard_Channel_2.Status/Error <-> AI Standard Channel 2/Status/Error
//     PlcTask Inputs/GVL_iXlinker.EtherCAT_Master_ELXxxxx.Beckhoff_ELXxxxx.A_0010_ELX3158_0000_0016.AI_Standard_Channel_3.Status/Error <-> AI Standard Channel 3/Status/Error
//     PlcTask Inputs/GVL_iXlinker.EtherCAT_Master_ELXxxxx.Beckhoff_ELXxxxx.A_0010_ELX3158_0000_0016.AI_Standard_Channel_4.Status/Error <-> AI Standard Channel 4/Status/Error
//     PlcTask Inputs/GVL_iXlinker.EtherCAT_Master_ELXxxxx.Beckhoff_ELXxxxx.A_0010_ELX3158_0000_0016.AI_Standard_Channel_5.Status/Error <-> AI Standard Channel 5/Status/Error
//     PlcTask Inputs/GVL_iXlinker.EtherCAT_Master_ELXxxxx.Beckhoff_ELXxxxx.A_0010_ELX3158_0000_0016.AI_Standard_Channel_6.Status/Error <-> AI Standard Channel 6/Status/Error
//     PlcTask Inputs/GVL_iXlinker.EtherCAT_Master_ELXxxxx.Beckhoff_ELXxxxx.A_0010_ELX3158_0000_0016.AI_Standard_Channel_7.Status/Error <-> AI Standard Channel 7/Status/Error
//     PlcTask Inputs/GVL_iXlinker.EtherCAT_Master_ELXxxxx.Beckhoff_ELXxxxx.A_0010_ELX3158_0000_0016.AI_Standard_Channel_8.Status/Error <-> AI Standard Channel 8/Status/Error
//     PlcTask Inputs/GVL_iXlinker.EtherCAT_Master_ELXxxxx.Beckhoff_ELXxxxx.A_0010_ELX3158_0000_0016.AI_Standard_Channel_1.Status/Sync_error <-> AI Standard Channel 1/Status/Sync error
//     PlcTask Inputs/GVL_iXlinker.EtherCAT_Master_ELXxxxx.Beckhoff_ELXxxxx.A_0010_ELX3158_0000_0016.AI_Standard_Channel_2.Status/Sync_error <-> AI Standard Channel 2/Status/Sync error
//     PlcTask Inputs/GVL_iXlinker.EtherCAT_Master_ELXxxxx.Beckhoff_ELXxxxx.A_0010_ELX3158_0000_0016.AI_Standard_Channel_3.Status/Sync_error <-> AI Standard Channel 3/Status/Sync error
//     PlcTask Inputs/GVL_iXlinker.EtherCAT_Master_ELXxxxx.Beckhoff_ELXxxxx.A_0010_ELX3158_0000_0016.AI_Standard_Channel_4.Status/Sync_error <-> AI Standard Channel 4/Status/Sync error
//     PlcTask Inputs/GVL_iXlinker.EtherCAT_Master_ELXxxxx.Beckhoff_ELXxxxx.A_0010_ELX3158_0000_0016.AI_Standard_Channel_5.Status/Sync_error <-> AI Standard Channel 5/Status/Sync error
//     PlcTask Inputs/GVL_iXlinker.EtherCAT_Master_ELXxxxx.Beckhoff_ELXxxxx.A_0010_ELX3158_0000_0016.AI_Standard_Channel_6.Status/Sync_error <-> AI Standard Channel 6/Status/Sync error
//     PlcTask Inputs/GVL_iXlinker.EtherCAT_Master_ELXxxxx.Beckhoff_ELXxxxx.A_0010_ELX3158_0000_0016.AI_Standard_Channel_7.Status/Sync_error <-> AI Standard Channel 7/Status/Sync error
//     PlcTask Inputs/GVL_iXlinker.EtherCAT_Master_ELXxxxx.Beckhoff_ELXxxxx.A_0010_ELX3158_0000_0016.AI_Standard_Channel_8.Status/Sync_error <-> AI Standard Channel 8/Status/Sync error
//     PlcTask Inputs/GVL_iXlinker.EtherCAT_Master_ELXxxxx.Beckhoff_ELXxxxx.A_0010_ELX3158_0000_0016.AI_Standard_Channel_1.Status/TxPDO_State <-> AI Standard Channel 1/Status/TxPDO State
//     PlcTask Inputs/GVL_iXlinker.EtherCAT_Master_ELXxxxx.Beckhoff_ELXxxxx.A_0010_ELX3158_0000_0016.AI_Standard_Channel_2.Status/TxPDO_State <-> AI Standard Channel 2/Status/TxPDO State
//     PlcTask Inputs/GVL_iXlinker.EtherCAT_Master_ELXxxxx.Beckhoff_ELXxxxx.A_0010_ELX3158_0000_0016.AI_Standard_Channel_3.Status/TxPDO_State <-> AI Standard Channel 3/Status/TxPDO State
//     PlcTask Inputs/GVL_iXlinker.EtherCAT_Master_ELXxxxx.Beckhoff_ELXxxxx.A_0010_ELX3158_0000_0016.AI_Standard_Channel_4.Status/TxPDO_State <-> AI Standard Channel 4/Status/TxPDO State
//     PlcTask Inputs/GVL_iXlinker.EtherCAT_Master_ELXxxxx.Beckhoff_ELXxxxx.A_0010_ELX3158_0000_0016.AI_Standard_Channel_5.Status/TxPDO_State <-> AI Standard Channel 5/Status/TxPDO State
//     PlcTask Inputs/GVL_iXlinker.EtherCAT_Master_ELXxxxx.Beckhoff_ELXxxxx.A_0010_ELX3158_0000_0016.AI_Standard_Channel_6.Status/TxPDO_State <-> AI Standard Channel 6/Status/TxPDO State
//     PlcTask Inputs/GVL_iXlinker.EtherCAT_Master_ELXxxxx.Beckhoff_ELXxxxx.A_0010_ELX3158_0000_0016.AI_Standard_Channel_7.Status/TxPDO_State <-> AI Standard Channel 7/Status/TxPDO State
//     PlcTask Inputs/GVL_iXlinker.EtherCAT_Master_ELXxxxx.Beckhoff_ELXxxxx.A_0010_ELX3158_0000_0016.AI_Standard_Channel_8.Status/TxPDO_State <-> AI Standard Channel 8/Status/TxPDO State
//     PlcTask Inputs/GVL_iXlinker.EtherCAT_Master_ELXxxxx.Beckhoff_ELXxxxx.A_0010_ELX3158_0000_0016.AI_Standard_Channel_1.Status/TxPDO_Toggle <-> AI Standard Channel 1/Status/TxPDO Toggle
//     PlcTask Inputs/GVL_iXlinker.EtherCAT_Master_ELXxxxx.Beckhoff_ELXxxxx.A_0010_ELX3158_0000_0016.AI_Standard_Channel_2.Status/TxPDO_Toggle <-> AI Standard Channel 2/Status/TxPDO Toggle
//     PlcTask Inputs/GVL_iXlinker.EtherCAT_Master_ELXxxxx.Beckhoff_ELXxxxx.A_0010_ELX3158_0000_0016.AI_Standard_Channel_3.Status/TxPDO_Toggle <-> AI Standard Channel 3/Status/TxPDO Toggle
//     PlcTask Inputs/GVL_iXlinker.EtherCAT_Master_ELXxxxx.Beckhoff_ELXxxxx.A_0010_ELX3158_0000_0016.AI_Standard_Channel_4.Status/TxPDO_Toggle <-> AI Standard Channel 4/Status/TxPDO Toggle
//     PlcTask Inputs/GVL_iXlinker.EtherCAT_Master_ELXxxxx.Beckhoff_ELXxxxx.A_0010_ELX3158_0000_0016.AI_Standard_Channel_5.Status/TxPDO_Toggle <-> AI Standard Channel 5/Status/TxPDO Toggle
//     PlcTask Inputs/GVL_iXlinker.EtherCAT_Master_ELXxxxx.Beckhoff_ELXxxxx.A_0010_ELX3158_0000_0016.AI_Standard_Channel_6.Status/TxPDO_Toggle <-> AI Standard Channel 6/Status/TxPDO Toggle
//     PlcTask Inputs/GVL_iXlinker.EtherCAT_Master_ELXxxxx.Beckhoff_ELXxxxx.A_0010_ELX3158_0000_0016.AI_Standard_Channel_7.Status/TxPDO_Toggle <-> AI Standard Channel 7/Status/TxPDO Toggle
//     PlcTask Inputs/GVL_iXlinker.EtherCAT_Master_ELXxxxx.Beckhoff_ELXxxxx.A_0010_ELX3158_0000_0016.AI_Standard_Channel_8.Status/TxPDO_Toggle <-> AI Standard Channel 8/Status/TxPDO Toggle
//     PlcTask Inputs/GVL_iXlinker.EtherCAT_Master_ELXxxxx.Beckhoff_ELXxxxx.A_0010_ELX3158_0000_0016.AI_Standard_Channel_1.Value <-> AI Standard Channel 1/Value
//     PlcTask Inputs/GVL_iXlinker.EtherCAT_Master_ELXxxxx.Beckhoff_ELXxxxx.A_0010_ELX3158_0000_0016.AI_Standard_Channel_2.Value <-> AI Standard Channel 2/Value
//     PlcTask Inputs/GVL_iXlinker.EtherCAT_Master_ELXxxxx.Beckhoff_ELXxxxx.A_0010_ELX3158_0000_0016.AI_Standard_Channel_3.Value <-> AI Standard Channel 3/Value
//     PlcTask Inputs/GVL_iXlinker.EtherCAT_Master_ELXxxxx.Beckhoff_ELXxxxx.A_0010_ELX3158_0000_0016.AI_Standard_Channel_4.Value <-> AI Standard Channel 4/Value
//     PlcTask Inputs/GVL_iXlinker.EtherCAT_Master_ELXxxxx.Beckhoff_ELXxxxx.A_0010_ELX3158_0000_0016.AI_Standard_Channel_5.Value <-> AI Standard Channel 5/Value
//     PlcTask Inputs/GVL_iXlinker.EtherCAT_Master_ELXxxxx.Beckhoff_ELXxxxx.A_0010_ELX3158_0000_0016.AI_Standard_Channel_6.Value <-> AI Standard Channel 6/Value
//     PlcTask Inputs/GVL_iXlinker.EtherCAT_Master_ELXxxxx.Beckhoff_ELXxxxx.A_0010_ELX3158_0000_0016.AI_Standard_Channel_7.Value <-> AI Standard Channel 7/Value
//     PlcTask Inputs/GVL_iXlinker.EtherCAT_Master_ELXxxxx.Beckhoff_ELXxxxx.A_0010_ELX3158_0000_0016.AI_Standard_Channel_8.Value <-> AI Standard Channel 8/Value
//     PlcTask Inputs/GVL_iXlinker.EtherCAT_Master_ELXxxxx.Beckhoff_ELXxxxx.A_0010_ELX3158_0000_0016.WcState.WcState <-> WcState/WcState
//     PlcTask Inputs/GVL_iXlinker.EtherCAT_Master_ELXxxxx.Beckhoff_ELXxxxx.A_0010_ELX3158_0000_0016.WcState.InputToggle <-> WcState/InputToggle
//     PlcTask Inputs/GVL_iXlinker.EtherCAT_Master_ELXxxxx.Beckhoff_ELXxxxx.A_0010_ELX3158_0000_0016.InfoData.AdsAddr <-> InfoData/AdsAddr
//     PlcTask Inputs/GVL_iXlinker.EtherCAT_Master_ELXxxxx.Beckhoff_ELXxxxx.A_0010_ELX3158_0000_0016.InfoData.State <-> InfoData/State
//   PLC/PLC Instance <-> EtherCAT Master ELXxxxx/Beckhoff ELXxxxx/A_0011(ELX3181-0000-0016)
//     PlcTask Inputs/GVL_iXlinker.EtherCAT_Master_ELXxxxx.Beckhoff_ELXxxxx.A_0011_ELX3181_0000_0016.Ch_1.Ch_1_Al_Inputs.Status/Underrange <-> Ch. 1/Ch. 1 Al Inputs/Status/Underrange
//     PlcTask Inputs/GVL_iXlinker.EtherCAT_Master_ELXxxxx.Beckhoff_ELXxxxx.A_0011_ELX3181_0000_0016.Ch_1.Ch_1_Al_Inputs.Status/Overrange <-> Ch. 1/Ch. 1 Al Inputs/Status/Overrange
//     PlcTask Inputs/GVL_iXlinker.EtherCAT_Master_ELXxxxx.Beckhoff_ELXxxxx.A_0011_ELX3181_0000_0016.Ch_1.Ch_1_Al_Inputs.Status/Limit_1 <-> Ch. 1/Ch. 1 Al Inputs/Status/Limit 1
//     PlcTask Inputs/GVL_iXlinker.EtherCAT_Master_ELXxxxx.Beckhoff_ELXxxxx.A_0011_ELX3181_0000_0016.Ch_1.Ch_1_Al_Inputs.Status/Limit_2 <-> Ch. 1/Ch. 1 Al Inputs/Status/Limit 2
//     PlcTask Inputs/GVL_iXlinker.EtherCAT_Master_ELXxxxx.Beckhoff_ELXxxxx.A_0011_ELX3181_0000_0016.Ch_1.Ch_1_Al_Inputs.Status/Error <-> Ch. 1/Ch. 1 Al Inputs/Status/Error
//     PlcTask Inputs/GVL_iXlinker.EtherCAT_Master_ELXxxxx.Beckhoff_ELXxxxx.A_0011_ELX3181_0000_0016.Ch_1.Ch_1_Al_Inputs.Status/Sync_Error <-> Ch. 1/Ch. 1 Al Inputs/Status/Sync Error
//     PlcTask Inputs/GVL_iXlinker.EtherCAT_Master_ELXxxxx.Beckhoff_ELXxxxx.A_0011_ELX3181_0000_0016.Ch_1.Ch_1_Al_Inputs.Status/TxPDO_State <-> Ch. 1/Ch. 1 Al Inputs/Status/TxPDO State
//     PlcTask Inputs/GVL_iXlinker.EtherCAT_Master_ELXxxxx.Beckhoff_ELXxxxx.A_0011_ELX3181_0000_0016.Ch_1.Ch_1_Al_Inputs.Status/TxPDO_Toggle <-> Ch. 1/Ch. 1 Al Inputs/Status/TxPDO Toggle
//     PlcTask Inputs/GVL_iXlinker.EtherCAT_Master_ELXxxxx.Beckhoff_ELXxxxx.A_0011_ELX3181_0000_0016.Ch_1.Ch_1_Al_Inputs.Value <-> Ch. 1/Ch. 1 Al Inputs/Value
//     PlcTask Inputs/GVL_iXlinker.EtherCAT_Master_ELXxxxx.Beckhoff_ELXxxxx.A_0011_ELX3181_0000_0016.WcState.WcState <-> WcState/WcState
//     PlcTask Inputs/GVL_iXlinker.EtherCAT_Master_ELXxxxx.Beckhoff_ELXxxxx.A_0011_ELX3181_0000_0016.WcState.InputToggle <-> WcState/InputToggle
//     PlcTask Inputs/GVL_iXlinker.EtherCAT_Master_ELXxxxx.Beckhoff_ELXxxxx.A_0011_ELX3181_0000_0016.InfoData.AdsAddr <-> InfoData/AdsAddr
//     PlcTask Inputs/GVL_iXlinker.EtherCAT_Master_ELXxxxx.Beckhoff_ELXxxxx.A_0011_ELX3181_0000_0016.InfoData.AoeNetId <-> InfoData/AoeNetId
//     PlcTask Inputs/GVL_iXlinker.EtherCAT_Master_ELXxxxx.Beckhoff_ELXxxxx.A_0011_ELX3181_0000_0016.InfoData.State <-> InfoData/State
//   PLC/PLC Instance <-> EtherCAT Master ELXxxxx/Beckhoff ELXxxxx/A_0012(ELX3181-0000-0017)
//     PlcTask Inputs/GVL_iXlinker.EtherCAT_Master_ELXxxxx.Beckhoff_ELXxxxx.A_0012_ELX3181_0000_0017.Ch_1.Ch_1_Al_Inputs.Status/Underrange <-> Ch. 1/Ch. 1 Al Inputs/Status/Underrange
//     PlcTask Inputs/GVL_iXlinker.EtherCAT_Master_ELXxxxx.Beckhoff_ELXxxxx.A_0012_ELX3181_0000_0017.Ch_1.Ch_1_Al_Inputs.Status/Overrange <-> Ch. 1/Ch. 1 Al Inputs/Status/Overrange
//     PlcTask Inputs/GVL_iXlinker.EtherCAT_Master_ELXxxxx.Beckhoff_ELXxxxx.A_0012_ELX3181_0000_0017.Ch_1.Ch_1_Al_Inputs.Status/Limit_1 <-> Ch. 1/Ch. 1 Al Inputs/Status/Limit 1
//     PlcTask Inputs/GVL_iXlinker.EtherCAT_Master_ELXxxxx.Beckhoff_ELXxxxx.A_0012_ELX3181_0000_0017.Ch_1.Ch_1_Al_Inputs.Status/Limit_2 <-> Ch. 1/Ch. 1 Al Inputs/Status/Limit 2
//     PlcTask Inputs/GVL_iXlinker.EtherCAT_Master_ELXxxxx.Beckhoff_ELXxxxx.A_0012_ELX3181_0000_0017.Ch_1.Ch_1_Al_Inputs.Status/Error <-> Ch. 1/Ch. 1 Al Inputs/Status/Error
//     PlcTask Inputs/GVL_iXlinker.EtherCAT_Master_ELXxxxx.Beckhoff_ELXxxxx.A_0012_ELX3181_0000_0017.Ch_1.Ch_1_Al_Inputs.Status/Sync_Error <-> Ch. 1/Ch. 1 Al Inputs/Status/Sync Error
//     PlcTask Inputs/GVL_iXlinker.EtherCAT_Master_ELXxxxx.Beckhoff_ELXxxxx.A_0012_ELX3181_0000_0017.Ch_1.Ch_1_Al_Inputs.Status/TxPDO_State <-> Ch. 1/Ch. 1 Al Inputs/Status/TxPDO State
//     PlcTask Inputs/GVL_iXlinker.EtherCAT_Master_ELXxxxx.Beckhoff_ELXxxxx.A_0012_ELX3181_0000_0017.Ch_1.Ch_1_Al_Inputs.Status/TxPDO_Toggle <-> Ch. 1/Ch. 1 Al Inputs/Status/TxPDO Toggle
//     PlcTask Inputs/GVL_iXlinker.EtherCAT_Master_ELXxxxx.Beckhoff_ELXxxxx.A_0012_ELX3181_0000_0017.Ch_1.Ch_1_Al_Inputs.Value <-> Ch. 1/Ch. 1 Al Inputs/Value
//     PlcTask Inputs/GVL_iXlinker.EtherCAT_Master_ELXxxxx.Beckhoff_ELXxxxx.A_0012_ELX3181_0000_0017.WcState.WcState <-> WcState/WcState
//     PlcTask Inputs/GVL_iXlinker.EtherCAT_Master_ELXxxxx.Beckhoff_ELXxxxx.A_0012_ELX3181_0000_0017.WcState.InputToggle <-> WcState/InputToggle
//     PlcTask Inputs/GVL_iXlinker.EtherCAT_Master_ELXxxxx.Beckhoff_ELXxxxx.A_0012_ELX3181_0000_0017.InfoData.AdsAddr <-> InfoData/AdsAddr
//     PlcTask Inputs/GVL_iXlinker.EtherCAT_Master_ELXxxxx.Beckhoff_ELXxxxx.A_0012_ELX3181_0000_0017.InfoData.AoeNetId <-> InfoData/AoeNetId
//     PlcTask Inputs/GVL_iXlinker.EtherCAT_Master_ELXxxxx.Beckhoff_ELXxxxx.A_0012_ELX3181_0000_0017.InfoData.State <-> InfoData/State
//   PLC/PLC Instance <-> EtherCAT Master ELXxxxx/Beckhoff ELXxxxx/A_0013(ELX3202-0000-0016)
//     PlcTask Inputs/GVL_iXlinker.EtherCAT_Master_ELXxxxx.Beckhoff_ELXxxxx.A_0013_ELX3202_0000_0016.RTD_Inputs_Channel_1.Status/Underrange <-> RTD Inputs Channel 1/Status/Underrange
//     PlcTask Inputs/GVL_iXlinker.EtherCAT_Master_ELXxxxx.Beckhoff_ELXxxxx.A_0013_ELX3202_0000_0016.RTD_Inputs_Channel_2.Status/Underrange <-> RTD Inputs Channel 2/Status/Underrange
//     PlcTask Inputs/GVL_iXlinker.EtherCAT_Master_ELXxxxx.Beckhoff_ELXxxxx.A_0013_ELX3202_0000_0016.RTD_Inputs_Channel_1.Status/Overrange <-> RTD Inputs Channel 1/Status/Overrange
//     PlcTask Inputs/GVL_iXlinker.EtherCAT_Master_ELXxxxx.Beckhoff_ELXxxxx.A_0013_ELX3202_0000_0016.RTD_Inputs_Channel_2.Status/Overrange <-> RTD Inputs Channel 2/Status/Overrange
//     PlcTask Inputs/GVL_iXlinker.EtherCAT_Master_ELXxxxx.Beckhoff_ELXxxxx.A_0013_ELX3202_0000_0016.RTD_Inputs_Channel_1.Status/Limit_1 <-> RTD Inputs Channel 1/Status/Limit 1
//     PlcTask Inputs/GVL_iXlinker.EtherCAT_Master_ELXxxxx.Beckhoff_ELXxxxx.A_0013_ELX3202_0000_0016.RTD_Inputs_Channel_1.Status/Limit_2 <-> RTD Inputs Channel 1/Status/Limit 2
//     PlcTask Inputs/GVL_iXlinker.EtherCAT_Master_ELXxxxx.Beckhoff_ELXxxxx.A_0013_ELX3202_0000_0016.RTD_Inputs_Channel_2.Status/Limit_1 <-> RTD Inputs Channel 2/Status/Limit 1
//     PlcTask Inputs/GVL_iXlinker.EtherCAT_Master_ELXxxxx.Beckhoff_ELXxxxx.A_0013_ELX3202_0000_0016.RTD_Inputs_Channel_2.Status/Limit_2 <-> RTD Inputs Channel 2/Status/Limit 2
//     PlcTask Inputs/GVL_iXlinker.EtherCAT_Master_ELXxxxx.Beckhoff_ELXxxxx.A_0013_ELX3202_0000_0016.RTD_Inputs_Channel_1.Status/Error <-> RTD Inputs Channel 1/Status/Error
//     PlcTask Inputs/GVL_iXlinker.EtherCAT_Master_ELXxxxx.Beckhoff_ELXxxxx.A_0013_ELX3202_0000_0016.RTD_Inputs_Channel_2.Status/Error <-> RTD Inputs Channel 2/Status/Error
//     PlcTask Inputs/GVL_iXlinker.EtherCAT_Master_ELXxxxx.Beckhoff_ELXxxxx.A_0013_ELX3202_0000_0016.RTD_Inputs_Channel_1.Status/TxPDO_State <-> RTD Inputs Channel 1/Status/TxPDO State
//     PlcTask Inputs/GVL_iXlinker.EtherCAT_Master_ELXxxxx.Beckhoff_ELXxxxx.A_0013_ELX3202_0000_0016.RTD_Inputs_Channel_2.Status/TxPDO_State <-> RTD Inputs Channel 2/Status/TxPDO State
//     PlcTask Inputs/GVL_iXlinker.EtherCAT_Master_ELXxxxx.Beckhoff_ELXxxxx.A_0013_ELX3202_0000_0016.RTD_Inputs_Channel_1.Status/TxPDO_Toggle <-> RTD Inputs Channel 1/Status/TxPDO Toggle
//     PlcTask Inputs/GVL_iXlinker.EtherCAT_Master_ELXxxxx.Beckhoff_ELXxxxx.A_0013_ELX3202_0000_0016.RTD_Inputs_Channel_2.Status/TxPDO_Toggle <-> RTD Inputs Channel 2/Status/TxPDO Toggle
//     PlcTask Inputs/GVL_iXlinker.EtherCAT_Master_ELXxxxx.Beckhoff_ELXxxxx.A_0013_ELX3202_0000_0016.RTD_Inputs_Channel_1.Value <-> RTD Inputs Channel 1/Value
//     PlcTask Inputs/GVL_iXlinker.EtherCAT_Master_ELXxxxx.Beckhoff_ELXxxxx.A_0013_ELX3202_0000_0016.RTD_Inputs_Channel_2.Value <-> RTD Inputs Channel 2/Value
//     PlcTask Inputs/GVL_iXlinker.EtherCAT_Master_ELXxxxx.Beckhoff_ELXxxxx.A_0013_ELX3202_0000_0016.WcState.WcState <-> WcState/WcState
//     PlcTask Inputs/GVL_iXlinker.EtherCAT_Master_ELXxxxx.Beckhoff_ELXxxxx.A_0013_ELX3202_0000_0016.WcState.InputToggle <-> WcState/InputToggle
//     PlcTask Inputs/GVL_iXlinker.EtherCAT_Master_ELXxxxx.Beckhoff_ELXxxxx.A_0013_ELX3202_0000_0016.InfoData.AdsAddr <-> InfoData/AdsAddr
//     PlcTask Inputs/GVL_iXlinker.EtherCAT_Master_ELXxxxx.Beckhoff_ELXxxxx.A_0013_ELX3202_0000_0016.InfoData.State <-> InfoData/State
//   PLC/PLC Instance <-> EtherCAT Master ELXxxxx/Beckhoff ELXxxxx/A_0014(ELX3202-0090-0016)
//     PlcTask Inputs/GVL_iXlinker.EtherCAT_Master_ELXxxxx.Beckhoff_ELXxxxx.A_0014_ELX3202_0090_0016.RTD_Inputs_Channel_1.Status/Underrange <-> RTD Inputs Channel 1/Status/Underrange
//     PlcTask Inputs/GVL_iXlinker.EtherCAT_Master_ELXxxxx.Beckhoff_ELXxxxx.A_0014_ELX3202_0090_0016.RTD_Inputs_Channel_2.Status/Underrange <-> RTD Inputs Channel 2/Status/Underrange
//     PlcTask Inputs/GVL_iXlinker.EtherCAT_Master_ELXxxxx.Beckhoff_ELXxxxx.A_0014_ELX3202_0090_0016.RTD_Inputs_Channel_1.Status/Overrange <-> RTD Inputs Channel 1/Status/Overrange
//     PlcTask Inputs/GVL_iXlinker.EtherCAT_Master_ELXxxxx.Beckhoff_ELXxxxx.A_0014_ELX3202_0090_0016.RTD_Inputs_Channel_2.Status/Overrange <-> RTD Inputs Channel 2/Status/Overrange
//     PlcTask Inputs/GVL_iXlinker.EtherCAT_Master_ELXxxxx.Beckhoff_ELXxxxx.A_0014_ELX3202_0090_0016.RTD_Inputs_Channel_1.Status/Limit_1 <-> RTD Inputs Channel 1/Status/Limit 1
//     PlcTask Inputs/GVL_iXlinker.EtherCAT_Master_ELXxxxx.Beckhoff_ELXxxxx.A_0014_ELX3202_0090_0016.RTD_Inputs_Channel_1.Status/Limit_2 <-> RTD Inputs Channel 1/Status/Limit 2
//     PlcTask Inputs/GVL_iXlinker.EtherCAT_Master_ELXxxxx.Beckhoff_ELXxxxx.A_0014_ELX3202_0090_0016.RTD_Inputs_Channel_2.Status/Limit_1 <-> RTD Inputs Channel 2/Status/Limit 1
//     PlcTask Inputs/GVL_iXlinker.EtherCAT_Master_ELXxxxx.Beckhoff_ELXxxxx.A_0014_ELX3202_0090_0016.RTD_Inputs_Channel_2.Status/Limit_2 <-> RTD Inputs Channel 2/Status/Limit 2
//     PlcTask Inputs/GVL_iXlinker.EtherCAT_Master_ELXxxxx.Beckhoff_ELXxxxx.A_0014_ELX3202_0090_0016.RTD_Inputs_Channel_1.Status/Error <-> RTD Inputs Channel 1/Status/Error
//     PlcTask Inputs/GVL_iXlinker.EtherCAT_Master_ELXxxxx.Beckhoff_ELXxxxx.A_0014_ELX3202_0090_0016.RTD_Inputs_Channel_2.Status/Error <-> RTD Inputs Channel 2/Status/Error
//     PlcTask Inputs/GVL_iXlinker.EtherCAT_Master_ELXxxxx.Beckhoff_ELXxxxx.A_0014_ELX3202_0090_0016.RTD_Inputs_Channel_1.Status/TxPDO_State <-> RTD Inputs Channel 1/Status/TxPDO State
//     PlcTask Inputs/GVL_iXlinker.EtherCAT_Master_ELXxxxx.Beckhoff_ELXxxxx.A_0014_ELX3202_0090_0016.RTD_Inputs_Channel_2.Status/TxPDO_State <-> RTD Inputs Channel 2/Status/TxPDO State
//     PlcTask Inputs/GVL_iXlinker.EtherCAT_Master_ELXxxxx.Beckhoff_ELXxxxx.A_0014_ELX3202_0090_0016.RTD_Inputs_Channel_1.Status/TxPDO_Toggle <-> RTD Inputs Channel 1/Status/TxPDO Toggle
//     PlcTask Inputs/GVL_iXlinker.EtherCAT_Master_ELXxxxx.Beckhoff_ELXxxxx.A_0014_ELX3202_0090_0016.RTD_Inputs_Channel_2.Status/TxPDO_Toggle <-> RTD Inputs Channel 2/Status/TxPDO Toggle
//     PlcTask Inputs/GVL_iXlinker.EtherCAT_Master_ELXxxxx.Beckhoff_ELXxxxx.A_0014_ELX3202_0090_0016.RTD_Inputs_Channel_1.Value <-> RTD Inputs Channel 1/Value
//     PlcTask Inputs/GVL_iXlinker.EtherCAT_Master_ELXxxxx.Beckhoff_ELXxxxx.A_0014_ELX3202_0090_0016.RTD_Inputs_Channel_2.Value <-> RTD Inputs Channel 2/Value
//     PlcTask Inputs/GVL_iXlinker.EtherCAT_Master_ELXxxxx.Beckhoff_ELXxxxx.A_0014_ELX3202_0090_0016.WcState.WcState <-> WcState/WcState
//     PlcTask Inputs/GVL_iXlinker.EtherCAT_Master_ELXxxxx.Beckhoff_ELXxxxx.A_0014_ELX3202_0090_0016.WcState.InputToggle <-> WcState/InputToggle
//     PlcTask Inputs/GVL_iXlinker.EtherCAT_Master_ELXxxxx.Beckhoff_ELXxxxx.A_0014_ELX3202_0090_0016.InfoData.AdsAddr <-> InfoData/AdsAddr
//     PlcTask Inputs/GVL_iXlinker.EtherCAT_Master_ELXxxxx.Beckhoff_ELXxxxx.A_0014_ELX3202_0090_0016.InfoData.State <-> InfoData/State
//   PLC/PLC Instance <-> EtherCAT Master ELXxxxx/Beckhoff ELXxxxx/A_0015(ELX3204-0000-0016)
//     PlcTask Inputs/GVL_iXlinker.EtherCAT_Master_ELXxxxx.Beckhoff_ELXxxxx.A_0015_ELX3204_0000_0016.RTD_Inputs_Channel_1.Status/Underrange <-> RTD Inputs Channel 1/Status/Underrange
//     PlcTask Inputs/GVL_iXlinker.EtherCAT_Master_ELXxxxx.Beckhoff_ELXxxxx.A_0015_ELX3204_0000_0016.RTD_Inputs_Channel_2.Status/Underrange <-> RTD Inputs Channel 2/Status/Underrange
//     PlcTask Inputs/GVL_iXlinker.EtherCAT_Master_ELXxxxx.Beckhoff_ELXxxxx.A_0015_ELX3204_0000_0016.RTD_Inputs_Channel_3.Status/Underrange <-> RTD Inputs Channel 3/Status/Underrange
//     PlcTask Inputs/GVL_iXlinker.EtherCAT_Master_ELXxxxx.Beckhoff_ELXxxxx.A_0015_ELX3204_0000_0016.RTD_Inputs_Channel_4.Status/Underrange <-> RTD Inputs Channel 4/Status/Underrange
//     PlcTask Inputs/GVL_iXlinker.EtherCAT_Master_ELXxxxx.Beckhoff_ELXxxxx.A_0015_ELX3204_0000_0016.RTD_Inputs_Channel_1.Status/Overrange <-> RTD Inputs Channel 1/Status/Overrange
//     PlcTask Inputs/GVL_iXlinker.EtherCAT_Master_ELXxxxx.Beckhoff_ELXxxxx.A_0015_ELX3204_0000_0016.RTD_Inputs_Channel_2.Status/Overrange <-> RTD Inputs Channel 2/Status/Overrange
//     PlcTask Inputs/GVL_iXlinker.EtherCAT_Master_ELXxxxx.Beckhoff_ELXxxxx.A_0015_ELX3204_0000_0016.RTD_Inputs_Channel_3.Status/Overrange <-> RTD Inputs Channel 3/Status/Overrange
//     PlcTask Inputs/GVL_iXlinker.EtherCAT_Master_ELXxxxx.Beckhoff_ELXxxxx.A_0015_ELX3204_0000_0016.RTD_Inputs_Channel_4.Status/Overrange <-> RTD Inputs Channel 4/Status/Overrange
//     PlcTask Inputs/GVL_iXlinker.EtherCAT_Master_ELXxxxx.Beckhoff_ELXxxxx.A_0015_ELX3204_0000_0016.RTD_Inputs_Channel_1.Status/Limit_1 <-> RTD Inputs Channel 1/Status/Limit 1
//     PlcTask Inputs/GVL_iXlinker.EtherCAT_Master_ELXxxxx.Beckhoff_ELXxxxx.A_0015_ELX3204_0000_0016.RTD_Inputs_Channel_1.Status/Limit_2 <-> RTD Inputs Channel 1/Status/Limit 2
//     PlcTask Inputs/GVL_iXlinker.EtherCAT_Master_ELXxxxx.Beckhoff_ELXxxxx.A_0015_ELX3204_0000_0016.RTD_Inputs_Channel_2.Status/Limit_1 <-> RTD Inputs Channel 2/Status/Limit 1
//     PlcTask Inputs/GVL_iXlinker.EtherCAT_Master_ELXxxxx.Beckhoff_ELXxxxx.A_0015_ELX3204_0000_0016.RTD_Inputs_Channel_2.Status/Limit_2 <-> RTD Inputs Channel 2/Status/Limit 2
//     PlcTask Inputs/GVL_iXlinker.EtherCAT_Master_ELXxxxx.Beckhoff_ELXxxxx.A_0015_ELX3204_0000_0016.RTD_Inputs_Channel_3.Status/Limit_1 <-> RTD Inputs Channel 3/Status/Limit 1
//     PlcTask Inputs/GVL_iXlinker.EtherCAT_Master_ELXxxxx.Beckhoff_ELXxxxx.A_0015_ELX3204_0000_0016.RTD_Inputs_Channel_3.Status/Limit_2 <-> RTD Inputs Channel 3/Status/Limit 2
//     PlcTask Inputs/GVL_iXlinker.EtherCAT_Master_ELXxxxx.Beckhoff_ELXxxxx.A_0015_ELX3204_0000_0016.RTD_Inputs_Channel_4.Status/Limit_1 <-> RTD Inputs Channel 4/Status/Limit 1
//     PlcTask Inputs/GVL_iXlinker.EtherCAT_Master_ELXxxxx.Beckhoff_ELXxxxx.A_0015_ELX3204_0000_0016.RTD_Inputs_Channel_4.Status/Limit_2 <-> RTD Inputs Channel 4/Status/Limit 2
//     PlcTask Inputs/GVL_iXlinker.EtherCAT_Master_ELXxxxx.Beckhoff_ELXxxxx.A_0015_ELX3204_0000_0016.RTD_Inputs_Channel_1.Status/Error <-> RTD Inputs Channel 1/Status/Error
//     PlcTask Inputs/GVL_iXlinker.EtherCAT_Master_ELXxxxx.Beckhoff_ELXxxxx.A_0015_ELX3204_0000_0016.RTD_Inputs_Channel_2.Status/Error <-> RTD Inputs Channel 2/Status/Error
//     PlcTask Inputs/GVL_iXlinker.EtherCAT_Master_ELXxxxx.Beckhoff_ELXxxxx.A_0015_ELX3204_0000_0016.RTD_Inputs_Channel_3.Status/Error <-> RTD Inputs Channel 3/Status/Error
//     PlcTask Inputs/GVL_iXlinker.EtherCAT_Master_ELXxxxx.Beckhoff_ELXxxxx.A_0015_ELX3204_0000_0016.RTD_Inputs_Channel_4.Status/Error <-> RTD Inputs Channel 4/Status/Error
//     PlcTask Inputs/GVL_iXlinker.EtherCAT_Master_ELXxxxx.Beckhoff_ELXxxxx.A_0015_ELX3204_0000_0016.RTD_Inputs_Channel_1.Status/TxPDO_State <-> RTD Inputs Channel 1/Status/TxPDO State
//     PlcTask Inputs/GVL_iXlinker.EtherCAT_Master_ELXxxxx.Beckhoff_ELXxxxx.A_0015_ELX3204_0000_0016.RTD_Inputs_Channel_2.Status/TxPDO_State <-> RTD Inputs Channel 2/Status/TxPDO State
//     PlcTask Inputs/GVL_iXlinker.EtherCAT_Master_ELXxxxx.Beckhoff_ELXxxxx.A_0015_ELX3204_0000_0016.RTD_Inputs_Channel_3.Status/TxPDO_State <-> RTD Inputs Channel 3/Status/TxPDO State
//     PlcTask Inputs/GVL_iXlinker.EtherCAT_Master_ELXxxxx.Beckhoff_ELXxxxx.A_0015_ELX3204_0000_0016.RTD_Inputs_Channel_4.Status/TxPDO_State <-> RTD Inputs Channel 4/Status/TxPDO State
//     PlcTask Inputs/GVL_iXlinker.EtherCAT_Master_ELXxxxx.Beckhoff_ELXxxxx.A_0015_ELX3204_0000_0016.RTD_Inputs_Channel_1.Status/TxPDO_Toggle <-> RTD Inputs Channel 1/Status/TxPDO Toggle
//     PlcTask Inputs/GVL_iXlinker.EtherCAT_Master_ELXxxxx.Beckhoff_ELXxxxx.A_0015_ELX3204_0000_0016.RTD_Inputs_Channel_2.Status/TxPDO_Toggle <-> RTD Inputs Channel 2/Status/TxPDO Toggle
//     PlcTask Inputs/GVL_iXlinker.EtherCAT_Master_ELXxxxx.Beckhoff_ELXxxxx.A_0015_ELX3204_0000_0016.RTD_Inputs_Channel_3.Status/TxPDO_Toggle <-> RTD Inputs Channel 3/Status/TxPDO Toggle
//     PlcTask Inputs/GVL_iXlinker.EtherCAT_Master_ELXxxxx.Beckhoff_ELXxxxx.A_0015_ELX3204_0000_0016.RTD_Inputs_Channel_4.Status/TxPDO_Toggle <-> RTD Inputs Channel 4/Status/TxPDO Toggle
//     PlcTask Inputs/GVL_iXlinker.EtherCAT_Master_ELXxxxx.Beckhoff_ELXxxxx.A_0015_ELX3204_0000_0016.RTD_Inputs_Channel_1.Value <-> RTD Inputs Channel 1/Value
//     PlcTask Inputs/GVL_iXlinker.EtherCAT_Master_ELXxxxx.Beckhoff_ELXxxxx.A_0015_ELX3204_0000_0016.RTD_Inputs_Channel_2.Value <-> RTD Inputs Channel 2/Value
//     PlcTask Inputs/GVL_iXlinker.EtherCAT_Master_ELXxxxx.Beckhoff_ELXxxxx.A_0015_ELX3204_0000_0016.RTD_Inputs_Channel_3.Value <-> RTD Inputs Channel 3/Value
//     PlcTask Inputs/GVL_iXlinker.EtherCAT_Master_ELXxxxx.Beckhoff_ELXxxxx.A_0015_ELX3204_0000_0016.RTD_Inputs_Channel_4.Value <-> RTD Inputs Channel 4/Value
//     PlcTask Inputs/GVL_iXlinker.EtherCAT_Master_ELXxxxx.Beckhoff_ELXxxxx.A_0015_ELX3204_0000_0016.WcState.WcState <-> WcState/WcState
//     PlcTask Inputs/GVL_iXlinker.EtherCAT_Master_ELXxxxx.Beckhoff_ELXxxxx.A_0015_ELX3204_0000_0016.WcState.InputToggle <-> WcState/InputToggle
//     PlcTask Inputs/GVL_iXlinker.EtherCAT_Master_ELXxxxx.Beckhoff_ELXxxxx.A_0015_ELX3204_0000_0016.InfoData.AdsAddr <-> InfoData/AdsAddr
//     PlcTask Inputs/GVL_iXlinker.EtherCAT_Master_ELXxxxx.Beckhoff_ELXxxxx.A_0015_ELX3204_0000_0016.InfoData.State <-> InfoData/State
//   PLC/PLC Instance <-> EtherCAT Master ELXxxxx/Beckhoff ELXxxxx/A_0016(ELX3204-0090-0016)
//     PlcTask Inputs/GVL_iXlinker.EtherCAT_Master_ELXxxxx.Beckhoff_ELXxxxx.A_0016_ELX3204_0090_0016.RTD_Inputs_Channel_1.Status/Underrange <-> RTD Inputs Channel 1/Status/Underrange
//     PlcTask Inputs/GVL_iXlinker.EtherCAT_Master_ELXxxxx.Beckhoff_ELXxxxx.A_0016_ELX3204_0090_0016.RTD_Inputs_Channel_2.Status/Underrange <-> RTD Inputs Channel 2/Status/Underrange
//     PlcTask Inputs/GVL_iXlinker.EtherCAT_Master_ELXxxxx.Beckhoff_ELXxxxx.A_0016_ELX3204_0090_0016.RTD_Inputs_Channel_3.Status/Underrange <-> RTD Inputs Channel 3/Status/Underrange
//     PlcTask Inputs/GVL_iXlinker.EtherCAT_Master_ELXxxxx.Beckhoff_ELXxxxx.A_0016_ELX3204_0090_0016.RTD_Inputs_Channel_4.Status/Underrange <-> RTD Inputs Channel 4/Status/Underrange
//     PlcTask Inputs/GVL_iXlinker.EtherCAT_Master_ELXxxxx.Beckhoff_ELXxxxx.A_0016_ELX3204_0090_0016.RTD_Inputs_Channel_1.Status/Overrange <-> RTD Inputs Channel 1/Status/Overrange
//     PlcTask Inputs/GVL_iXlinker.EtherCAT_Master_ELXxxxx.Beckhoff_ELXxxxx.A_0016_ELX3204_0090_0016.RTD_Inputs_Channel_2.Status/Overrange <-> RTD Inputs Channel 2/Status/Overrange
//     PlcTask Inputs/GVL_iXlinker.EtherCAT_Master_ELXxxxx.Beckhoff_ELXxxxx.A_0016_ELX3204_0090_0016.RTD_Inputs_Channel_3.Status/Overrange <-> RTD Inputs Channel 3/Status/Overrange
//     PlcTask Inputs/GVL_iXlinker.EtherCAT_Master_ELXxxxx.Beckhoff_ELXxxxx.A_0016_ELX3204_0090_0016.RTD_Inputs_Channel_4.Status/Overrange <-> RTD Inputs Channel 4/Status/Overrange
//     PlcTask Inputs/GVL_iXlinker.EtherCAT_Master_ELXxxxx.Beckhoff_ELXxxxx.A_0016_ELX3204_0090_0016.RTD_Inputs_Channel_1.Status/Limit_1 <-> RTD Inputs Channel 1/Status/Limit 1
//     PlcTask Inputs/GVL_iXlinker.EtherCAT_Master_ELXxxxx.Beckhoff_ELXxxxx.A_0016_ELX3204_0090_0016.RTD_Inputs_Channel_1.Status/Limit_2 <-> RTD Inputs Channel 1/Status/Limit 2
//     PlcTask Inputs/GVL_iXlinker.EtherCAT_Master_ELXxxxx.Beckhoff_ELXxxxx.A_0016_ELX3204_0090_0016.RTD_Inputs_Channel_2.Status/Limit_1 <-> RTD Inputs Channel 2/Status/Limit 1
//     PlcTask Inputs/GVL_iXlinker.EtherCAT_Master_ELXxxxx.Beckhoff_ELXxxxx.A_0016_ELX3204_0090_0016.RTD_Inputs_Channel_2.Status/Limit_2 <-> RTD Inputs Channel 2/Status/Limit 2
//     PlcTask Inputs/GVL_iXlinker.EtherCAT_Master_ELXxxxx.Beckhoff_ELXxxxx.A_0016_ELX3204_0090_0016.RTD_Inputs_Channel_3.Status/Limit_1 <-> RTD Inputs Channel 3/Status/Limit 1
//     PlcTask Inputs/GVL_iXlinker.EtherCAT_Master_ELXxxxx.Beckhoff_ELXxxxx.A_0016_ELX3204_0090_0016.RTD_Inputs_Channel_3.Status/Limit_2 <-> RTD Inputs Channel 3/Status/Limit 2
//     PlcTask Inputs/GVL_iXlinker.EtherCAT_Master_ELXxxxx.Beckhoff_ELXxxxx.A_0016_ELX3204_0090_0016.RTD_Inputs_Channel_4.Status/Limit_1 <-> RTD Inputs Channel 4/Status/Limit 1
//     PlcTask Inputs/GVL_iXlinker.EtherCAT_Master_ELXxxxx.Beckhoff_ELXxxxx.A_0016_ELX3204_0090_0016.RTD_Inputs_Channel_4.Status/Limit_2 <-> RTD Inputs Channel 4/Status/Limit 2
//     PlcTask Inputs/GVL_iXlinker.EtherCAT_Master_ELXxxxx.Beckhoff_ELXxxxx.A_0016_ELX3204_0090_0016.RTD_Inputs_Channel_1.Status/Error <-> RTD Inputs Channel 1/Status/Error
//     PlcTask Inputs/GVL_iXlinker.EtherCAT_Master_ELXxxxx.Beckhoff_ELXxxxx.A_0016_ELX3204_0090_0016.RTD_Inputs_Channel_2.Status/Error <-> RTD Inputs Channel 2/Status/Error
//     PlcTask Inputs/GVL_iXlinker.EtherCAT_Master_ELXxxxx.Beckhoff_ELXxxxx.A_0016_ELX3204_0090_0016.RTD_Inputs_Channel_3.Status/Error <-> RTD Inputs Channel 3/Status/Error
//     PlcTask Inputs/GVL_iXlinker.EtherCAT_Master_ELXxxxx.Beckhoff_ELXxxxx.A_0016_ELX3204_0090_0016.RTD_Inputs_Channel_4.Status/Error <-> RTD Inputs Channel 4/Status/Error
//     PlcTask Inputs/GVL_iXlinker.EtherCAT_Master_ELXxxxx.Beckhoff_ELXxxxx.A_0016_ELX3204_0090_0016.RTD_Inputs_Channel_1.Status/TxPDO_State <-> RTD Inputs Channel 1/Status/TxPDO State
//     PlcTask Inputs/GVL_iXlinker.EtherCAT_Master_ELXxxxx.Beckhoff_ELXxxxx.A_0016_ELX3204_0090_0016.RTD_Inputs_Channel_2.Status/TxPDO_State <-> RTD Inputs Channel 2/Status/TxPDO State
//     PlcTask Inputs/GVL_iXlinker.EtherCAT_Master_ELXxxxx.Beckhoff_ELXxxxx.A_0016_ELX3204_0090_0016.RTD_Inputs_Channel_3.Status/TxPDO_State <-> RTD Inputs Channel 3/Status/TxPDO State
//     PlcTask Inputs/GVL_iXlinker.EtherCAT_Master_ELXxxxx.Beckhoff_ELXxxxx.A_0016_ELX3204_0090_0016.RTD_Inputs_Channel_4.Status/TxPDO_State <-> RTD Inputs Channel 4/Status/TxPDO State
//     PlcTask Inputs/GVL_iXlinker.EtherCAT_Master_ELXxxxx.Beckhoff_ELXxxxx.A_0016_ELX3204_0090_0016.RTD_Inputs_Channel_1.Status/TxPDO_Toggle <-> RTD Inputs Channel 1/Status/TxPDO Toggle
//     PlcTask Inputs/GVL_iXlinker.EtherCAT_Master_ELXxxxx.Beckhoff_ELXxxxx.A_0016_ELX3204_0090_0016.RTD_Inputs_Channel_2.Status/TxPDO_Toggle <-> RTD Inputs Channel 2/Status/TxPDO Toggle
//     PlcTask Inputs/GVL_iXlinker.EtherCAT_Master_ELXxxxx.Beckhoff_ELXxxxx.A_0016_ELX3204_0090_0016.RTD_Inputs_Channel_3.Status/TxPDO_Toggle <-> RTD Inputs Channel 3/Status/TxPDO Toggle
//     PlcTask Inputs/GVL_iXlinker.EtherCAT_Master_ELXxxxx.Beckhoff_ELXxxxx.A_0016_ELX3204_0090_0016.RTD_Inputs_Channel_4.Status/TxPDO_Toggle <-> RTD Inputs Channel 4/Status/TxPDO Toggle
//     PlcTask Inputs/GVL_iXlinker.EtherCAT_Master_ELXxxxx.Beckhoff_ELXxxxx.A_0016_ELX3204_0090_0016.RTD_Inputs_Channel_1.Value <-> RTD Inputs Channel 1/Value
//     PlcTask Inputs/GVL_iXlinker.EtherCAT_Master_ELXxxxx.Beckhoff_ELXxxxx.A_0016_ELX3204_0090_0016.RTD_Inputs_Channel_2.Value <-> RTD Inputs Channel 2/Value
//     PlcTask Inputs/GVL_iXlinker.EtherCAT_Master_ELXxxxx.Beckhoff_ELXxxxx.A_0016_ELX3204_0090_0016.RTD_Inputs_Channel_3.Value <-> RTD Inputs Channel 3/Value
//     PlcTask Inputs/GVL_iXlinker.EtherCAT_Master_ELXxxxx.Beckhoff_ELXxxxx.A_0016_ELX3204_0090_0016.RTD_Inputs_Channel_4.Value <-> RTD Inputs Channel 4/Value
//     PlcTask Inputs/GVL_iXlinker.EtherCAT_Master_ELXxxxx.Beckhoff_ELXxxxx.A_0016_ELX3204_0090_0016.WcState.WcState <-> WcState/WcState
//     PlcTask Inputs/GVL_iXlinker.EtherCAT_Master_ELXxxxx.Beckhoff_ELXxxxx.A_0016_ELX3204_0090_0016.WcState.InputToggle <-> WcState/InputToggle
//     PlcTask Inputs/GVL_iXlinker.EtherCAT_Master_ELXxxxx.Beckhoff_ELXxxxx.A_0016_ELX3204_0090_0016.InfoData.AdsAddr <-> InfoData/AdsAddr
//     PlcTask Inputs/GVL_iXlinker.EtherCAT_Master_ELXxxxx.Beckhoff_ELXxxxx.A_0016_ELX3204_0090_0016.InfoData.State <-> InfoData/State
//   PLC/PLC Instance <-> EtherCAT Master ELXxxxx/Beckhoff ELXxxxx/A_0017(ELX3252-0000-0016)
//     PlcTask Inputs/GVL_iXlinker.EtherCAT_Master_ELXxxxx.Beckhoff_ELXxxxx.A_0017_ELX3252_0000_0016.AI_Standard_Channel_1.Status/Limit_1 <-> AI Standard Channel 1/Status/Limit 1
//     PlcTask Inputs/GVL_iXlinker.EtherCAT_Master_ELXxxxx.Beckhoff_ELXxxxx.A_0017_ELX3252_0000_0016.AI_Standard_Channel_1.Status/Limit_2 <-> AI Standard Channel 1/Status/Limit 2
//     PlcTask Inputs/GVL_iXlinker.EtherCAT_Master_ELXxxxx.Beckhoff_ELXxxxx.A_0017_ELX3252_0000_0016.AI_Standard_Channel_2.Status/Limit_1 <-> AI Standard Channel 2/Status/Limit 1
//     PlcTask Inputs/GVL_iXlinker.EtherCAT_Master_ELXxxxx.Beckhoff_ELXxxxx.A_0017_ELX3252_0000_0016.AI_Standard_Channel_2.Status/Limit_2 <-> AI Standard Channel 2/Status/Limit 2
//     PlcTask Inputs/GVL_iXlinker.EtherCAT_Master_ELXxxxx.Beckhoff_ELXxxxx.A_0017_ELX3252_0000_0016.AI_Standard_Channel_1.Status/Error <-> AI Standard Channel 1/Status/Error
//     PlcTask Inputs/GVL_iXlinker.EtherCAT_Master_ELXxxxx.Beckhoff_ELXxxxx.A_0017_ELX3252_0000_0016.AI_Standard_Channel_2.Status/Error <-> AI Standard Channel 2/Status/Error
//     PlcTask Inputs/GVL_iXlinker.EtherCAT_Master_ELXxxxx.Beckhoff_ELXxxxx.A_0017_ELX3252_0000_0016.AI_Standard_Channel_1.Status/TxPDO_State <-> AI Standard Channel 1/Status/TxPDO State
//     PlcTask Inputs/GVL_iXlinker.EtherCAT_Master_ELXxxxx.Beckhoff_ELXxxxx.A_0017_ELX3252_0000_0016.AI_Standard_Channel_2.Status/TxPDO_State <-> AI Standard Channel 2/Status/TxPDO State
//     PlcTask Inputs/GVL_iXlinker.EtherCAT_Master_ELXxxxx.Beckhoff_ELXxxxx.A_0017_ELX3252_0000_0016.AI_Standard_Channel_1.Status/TxPDO_Toggle <-> AI Standard Channel 1/Status/TxPDO Toggle
//     PlcTask Inputs/GVL_iXlinker.EtherCAT_Master_ELXxxxx.Beckhoff_ELXxxxx.A_0017_ELX3252_0000_0016.AI_Standard_Channel_2.Status/TxPDO_Toggle <-> AI Standard Channel 2/Status/TxPDO Toggle
//     PlcTask Inputs/GVL_iXlinker.EtherCAT_Master_ELXxxxx.Beckhoff_ELXxxxx.A_0017_ELX3252_0000_0016.AI_Standard_Channel_1.Value <-> AI Standard Channel 1/Value
//     PlcTask Inputs/GVL_iXlinker.EtherCAT_Master_ELXxxxx.Beckhoff_ELXxxxx.A_0017_ELX3252_0000_0016.AI_Standard_Channel_2.Value <-> AI Standard Channel 2/Value
//     PlcTask Inputs/GVL_iXlinker.EtherCAT_Master_ELXxxxx.Beckhoff_ELXxxxx.A_0017_ELX3252_0000_0016.WcState.WcState <-> WcState/WcState
//     PlcTask Inputs/GVL_iXlinker.EtherCAT_Master_ELXxxxx.Beckhoff_ELXxxxx.A_0017_ELX3252_0000_0016.WcState.InputToggle <-> WcState/InputToggle
//     PlcTask Inputs/GVL_iXlinker.EtherCAT_Master_ELXxxxx.Beckhoff_ELXxxxx.A_0017_ELX3252_0000_0016.InfoData.AdsAddr <-> InfoData/AdsAddr
//     PlcTask Inputs/GVL_iXlinker.EtherCAT_Master_ELXxxxx.Beckhoff_ELXxxxx.A_0017_ELX3252_0000_0016.InfoData.State <-> InfoData/State
//   PLC/PLC Instance <-> EtherCAT Master ELXxxxx/Beckhoff ELXxxxx/A_0018(ELX3312-0000-0016)
//     PlcTask Inputs/GVL_iXlinker.EtherCAT_Master_ELXxxxx.Beckhoff_ELXxxxx.A_0018_ELX3312_0000_0016.TC_Inputs_Channel_1.Status/Underrange <-> TC Inputs Channel 1/Status/Underrange
//     PlcTask Inputs/GVL_iXlinker.EtherCAT_Master_ELXxxxx.Beckhoff_ELXxxxx.A_0018_ELX3312_0000_0016.TC_Inputs_Channel_2.Status/Underrange <-> TC Inputs Channel 2/Status/Underrange
//     PlcTask Inputs/GVL_iXlinker.EtherCAT_Master_ELXxxxx.Beckhoff_ELXxxxx.A_0018_ELX3312_0000_0016.TC_Inputs_Channel_1.Status/Overrange <-> TC Inputs Channel 1/Status/Overrange
//     PlcTask Inputs/GVL_iXlinker.EtherCAT_Master_ELXxxxx.Beckhoff_ELXxxxx.A_0018_ELX3312_0000_0016.TC_Inputs_Channel_2.Status/Overrange <-> TC Inputs Channel 2/Status/Overrange
//     PlcTask Inputs/GVL_iXlinker.EtherCAT_Master_ELXxxxx.Beckhoff_ELXxxxx.A_0018_ELX3312_0000_0016.TC_Inputs_Channel_1.Status/Limit_1 <-> TC Inputs Channel 1/Status/Limit 1
//     PlcTask Inputs/GVL_iXlinker.EtherCAT_Master_ELXxxxx.Beckhoff_ELXxxxx.A_0018_ELX3312_0000_0016.TC_Inputs_Channel_1.Status/Limit_2 <-> TC Inputs Channel 1/Status/Limit 2
//     PlcTask Inputs/GVL_iXlinker.EtherCAT_Master_ELXxxxx.Beckhoff_ELXxxxx.A_0018_ELX3312_0000_0016.TC_Inputs_Channel_2.Status/Limit_1 <-> TC Inputs Channel 2/Status/Limit 1
//     PlcTask Inputs/GVL_iXlinker.EtherCAT_Master_ELXxxxx.Beckhoff_ELXxxxx.A_0018_ELX3312_0000_0016.TC_Inputs_Channel_2.Status/Limit_2 <-> TC Inputs Channel 2/Status/Limit 2
//     PlcTask Inputs/GVL_iXlinker.EtherCAT_Master_ELXxxxx.Beckhoff_ELXxxxx.A_0018_ELX3312_0000_0016.TC_Inputs_Channel_1.Status/Error <-> TC Inputs Channel 1/Status/Error
//     PlcTask Inputs/GVL_iXlinker.EtherCAT_Master_ELXxxxx.Beckhoff_ELXxxxx.A_0018_ELX3312_0000_0016.TC_Inputs_Channel_2.Status/Error <-> TC Inputs Channel 2/Status/Error
//     PlcTask Inputs/GVL_iXlinker.EtherCAT_Master_ELXxxxx.Beckhoff_ELXxxxx.A_0018_ELX3312_0000_0016.TC_Inputs_Channel_1.Status/TxPDO_State <-> TC Inputs Channel 1/Status/TxPDO State
//     PlcTask Inputs/GVL_iXlinker.EtherCAT_Master_ELXxxxx.Beckhoff_ELXxxxx.A_0018_ELX3312_0000_0016.TC_Inputs_Channel_2.Status/TxPDO_State <-> TC Inputs Channel 2/Status/TxPDO State
//     PlcTask Inputs/GVL_iXlinker.EtherCAT_Master_ELXxxxx.Beckhoff_ELXxxxx.A_0018_ELX3312_0000_0016.TC_Inputs_Channel_1.Status/TxPDO_Toggle <-> TC Inputs Channel 1/Status/TxPDO Toggle
//     PlcTask Inputs/GVL_iXlinker.EtherCAT_Master_ELXxxxx.Beckhoff_ELXxxxx.A_0018_ELX3312_0000_0016.TC_Inputs_Channel_2.Status/TxPDO_Toggle <-> TC Inputs Channel 2/Status/TxPDO Toggle
//     PlcTask Inputs/GVL_iXlinker.EtherCAT_Master_ELXxxxx.Beckhoff_ELXxxxx.A_0018_ELX3312_0000_0016.TC_Inputs_Channel_1.Value <-> TC Inputs Channel 1/Value
//     PlcTask Inputs/GVL_iXlinker.EtherCAT_Master_ELXxxxx.Beckhoff_ELXxxxx.A_0018_ELX3312_0000_0016.TC_Inputs_Channel_2.Value <-> TC Inputs Channel 2/Value
//     PlcTask Inputs/GVL_iXlinker.EtherCAT_Master_ELXxxxx.Beckhoff_ELXxxxx.A_0018_ELX3312_0000_0016.WcState.WcState <-> WcState/WcState
//     PlcTask Inputs/GVL_iXlinker.EtherCAT_Master_ELXxxxx.Beckhoff_ELXxxxx.A_0018_ELX3312_0000_0016.WcState.InputToggle <-> WcState/InputToggle
//     PlcTask Inputs/GVL_iXlinker.EtherCAT_Master_ELXxxxx.Beckhoff_ELXxxxx.A_0018_ELX3312_0000_0016.InfoData.AdsAddr <-> InfoData/AdsAddr
//     PlcTask Inputs/GVL_iXlinker.EtherCAT_Master_ELXxxxx.Beckhoff_ELXxxxx.A_0018_ELX3312_0000_0016.InfoData.State <-> InfoData/State
//   PLC/PLC Instance <-> EtherCAT Master ELXxxxx/Beckhoff ELXxxxx/A_0019(ELX3312-0090-0016)
//     PlcTask Inputs/GVL_iXlinker.EtherCAT_Master_ELXxxxx.Beckhoff_ELXxxxx.A_0019_ELX3312_0090_0016.TC_Inputs_Channel_1.Status/Underrange <-> TC Inputs Channel 1/Status/Underrange
//     PlcTask Inputs/GVL_iXlinker.EtherCAT_Master_ELXxxxx.Beckhoff_ELXxxxx.A_0019_ELX3312_0090_0016.TC_Inputs_Channel_2.Status/Underrange <-> TC Inputs Channel 2/Status/Underrange
//     PlcTask Inputs/GVL_iXlinker.EtherCAT_Master_ELXxxxx.Beckhoff_ELXxxxx.A_0019_ELX3312_0090_0016.TC_Inputs_Channel_1.Status/Overrange <-> TC Inputs Channel 1/Status/Overrange
//     PlcTask Inputs/GVL_iXlinker.EtherCAT_Master_ELXxxxx.Beckhoff_ELXxxxx.A_0019_ELX3312_0090_0016.TC_Inputs_Channel_2.Status/Overrange <-> TC Inputs Channel 2/Status/Overrange
//     PlcTask Inputs/GVL_iXlinker.EtherCAT_Master_ELXxxxx.Beckhoff_ELXxxxx.A_0019_ELX3312_0090_0016.TC_Inputs_Channel_1.Status/Limit_1 <-> TC Inputs Channel 1/Status/Limit 1
//     PlcTask Inputs/GVL_iXlinker.EtherCAT_Master_ELXxxxx.Beckhoff_ELXxxxx.A_0019_ELX3312_0090_0016.TC_Inputs_Channel_1.Status/Limit_2 <-> TC Inputs Channel 1/Status/Limit 2
//     PlcTask Inputs/GVL_iXlinker.EtherCAT_Master_ELXxxxx.Beckhoff_ELXxxxx.A_0019_ELX3312_0090_0016.TC_Inputs_Channel_2.Status/Limit_1 <-> TC Inputs Channel 2/Status/Limit 1
//     PlcTask Inputs/GVL_iXlinker.EtherCAT_Master_ELXxxxx.Beckhoff_ELXxxxx.A_0019_ELX3312_0090_0016.TC_Inputs_Channel_2.Status/Limit_2 <-> TC Inputs Channel 2/Status/Limit 2
//     PlcTask Inputs/GVL_iXlinker.EtherCAT_Master_ELXxxxx.Beckhoff_ELXxxxx.A_0019_ELX3312_0090_0016.TC_Inputs_Channel_1.Status/Error <-> TC Inputs Channel 1/Status/Error
//     PlcTask Inputs/GVL_iXlinker.EtherCAT_Master_ELXxxxx.Beckhoff_ELXxxxx.A_0019_ELX3312_0090_0016.TC_Inputs_Channel_2.Status/Error <-> TC Inputs Channel 2/Status/Error
//     PlcTask Inputs/GVL_iXlinker.EtherCAT_Master_ELXxxxx.Beckhoff_ELXxxxx.A_0019_ELX3312_0090_0016.TC_Inputs_Channel_1.Status/TxPDO_State <-> TC Inputs Channel 1/Status/TxPDO State
//     PlcTask Inputs/GVL_iXlinker.EtherCAT_Master_ELXxxxx.Beckhoff_ELXxxxx.A_0019_ELX3312_0090_0016.TC_Inputs_Channel_2.Status/TxPDO_State <-> TC Inputs Channel 2/Status/TxPDO State
//     PlcTask Inputs/GVL_iXlinker.EtherCAT_Master_ELXxxxx.Beckhoff_ELXxxxx.A_0019_ELX3312_0090_0016.TC_Inputs_Channel_1.Status/TxPDO_Toggle <-> TC Inputs Channel 1/Status/TxPDO Toggle
//     PlcTask Inputs/GVL_iXlinker.EtherCAT_Master_ELXxxxx.Beckhoff_ELXxxxx.A_0019_ELX3312_0090_0016.TC_Inputs_Channel_2.Status/TxPDO_Toggle <-> TC Inputs Channel 2/Status/TxPDO Toggle
//     PlcTask Inputs/GVL_iXlinker.EtherCAT_Master_ELXxxxx.Beckhoff_ELXxxxx.A_0019_ELX3312_0090_0016.TC_Inputs_Channel_1.Value <-> TC Inputs Channel 1/Value
//     PlcTask Inputs/GVL_iXlinker.EtherCAT_Master_ELXxxxx.Beckhoff_ELXxxxx.A_0019_ELX3312_0090_0016.TC_Inputs_Channel_2.Value <-> TC Inputs Channel 2/Value
//     PlcTask Inputs/GVL_iXlinker.EtherCAT_Master_ELXxxxx.Beckhoff_ELXxxxx.A_0019_ELX3312_0090_0016.WcState.WcState <-> WcState/WcState
//     PlcTask Inputs/GVL_iXlinker.EtherCAT_Master_ELXxxxx.Beckhoff_ELXxxxx.A_0019_ELX3312_0090_0016.WcState.InputToggle <-> WcState/InputToggle
//     PlcTask Inputs/GVL_iXlinker.EtherCAT_Master_ELXxxxx.Beckhoff_ELXxxxx.A_0019_ELX3312_0090_0016.InfoData.AdsAddr <-> InfoData/AdsAddr
//     PlcTask Inputs/GVL_iXlinker.EtherCAT_Master_ELXxxxx.Beckhoff_ELXxxxx.A_0019_ELX3312_0090_0016.InfoData.State <-> InfoData/State
//   PLC/PLC Instance <-> EtherCAT Master ELXxxxx/Beckhoff ELXxxxx/A_0020(ELX3314-0000-0016)
//     PlcTask Inputs/GVL_iXlinker.EtherCAT_Master_ELXxxxx.Beckhoff_ELXxxxx.A_0020_ELX3314_0000_0016.TC_Inputs_Channel_1.Status/Underrange <-> TC Inputs Channel 1/Status/Underrange
//     PlcTask Inputs/GVL_iXlinker.EtherCAT_Master_ELXxxxx.Beckhoff_ELXxxxx.A_0020_ELX3314_0000_0016.TC_Inputs_Channel_2.Status/Underrange <-> TC Inputs Channel 2/Status/Underrange
//     PlcTask Inputs/GVL_iXlinker.EtherCAT_Master_ELXxxxx.Beckhoff_ELXxxxx.A_0020_ELX3314_0000_0016.TC_Inputs_Channel_3.Status/Underrange <-> TC Inputs Channel 3/Status/Underrange
//     PlcTask Inputs/GVL_iXlinker.EtherCAT_Master_ELXxxxx.Beckhoff_ELXxxxx.A_0020_ELX3314_0000_0016.TC_Inputs_Channel_4.Status/Underrange <-> TC Inputs Channel 4/Status/Underrange
//     PlcTask Inputs/GVL_iXlinker.EtherCAT_Master_ELXxxxx.Beckhoff_ELXxxxx.A_0020_ELX3314_0000_0016.TC_Inputs_Channel_1.Status/Overrange <-> TC Inputs Channel 1/Status/Overrange
//     PlcTask Inputs/GVL_iXlinker.EtherCAT_Master_ELXxxxx.Beckhoff_ELXxxxx.A_0020_ELX3314_0000_0016.TC_Inputs_Channel_2.Status/Overrange <-> TC Inputs Channel 2/Status/Overrange
//     PlcTask Inputs/GVL_iXlinker.EtherCAT_Master_ELXxxxx.Beckhoff_ELXxxxx.A_0020_ELX3314_0000_0016.TC_Inputs_Channel_3.Status/Overrange <-> TC Inputs Channel 3/Status/Overrange
//     PlcTask Inputs/GVL_iXlinker.EtherCAT_Master_ELXxxxx.Beckhoff_ELXxxxx.A_0020_ELX3314_0000_0016.TC_Inputs_Channel_4.Status/Overrange <-> TC Inputs Channel 4/Status/Overrange
//     PlcTask Inputs/GVL_iXlinker.EtherCAT_Master_ELXxxxx.Beckhoff_ELXxxxx.A_0020_ELX3314_0000_0016.TC_Inputs_Channel_1.Status/Limit_1 <-> TC Inputs Channel 1/Status/Limit 1
//     PlcTask Inputs/GVL_iXlinker.EtherCAT_Master_ELXxxxx.Beckhoff_ELXxxxx.A_0020_ELX3314_0000_0016.TC_Inputs_Channel_1.Status/Limit_2 <-> TC Inputs Channel 1/Status/Limit 2
//     PlcTask Inputs/GVL_iXlinker.EtherCAT_Master_ELXxxxx.Beckhoff_ELXxxxx.A_0020_ELX3314_0000_0016.TC_Inputs_Channel_2.Status/Limit_1 <-> TC Inputs Channel 2/Status/Limit 1
//     PlcTask Inputs/GVL_iXlinker.EtherCAT_Master_ELXxxxx.Beckhoff_ELXxxxx.A_0020_ELX3314_0000_0016.TC_Inputs_Channel_2.Status/Limit_2 <-> TC Inputs Channel 2/Status/Limit 2
//     PlcTask Inputs/GVL_iXlinker.EtherCAT_Master_ELXxxxx.Beckhoff_ELXxxxx.A_0020_ELX3314_0000_0016.TC_Inputs_Channel_3.Status/Limit_1 <-> TC Inputs Channel 3/Status/Limit 1
//     PlcTask Inputs/GVL_iXlinker.EtherCAT_Master_ELXxxxx.Beckhoff_ELXxxxx.A_0020_ELX3314_0000_0016.TC_Inputs_Channel_3.Status/Limit_2 <-> TC Inputs Channel 3/Status/Limit 2
//     PlcTask Inputs/GVL_iXlinker.EtherCAT_Master_ELXxxxx.Beckhoff_ELXxxxx.A_0020_ELX3314_0000_0016.TC_Inputs_Channel_4.Status/Limit_1 <-> TC Inputs Channel 4/Status/Limit 1
//     PlcTask Inputs/GVL_iXlinker.EtherCAT_Master_ELXxxxx.Beckhoff_ELXxxxx.A_0020_ELX3314_0000_0016.TC_Inputs_Channel_4.Status/Limit_2 <-> TC Inputs Channel 4/Status/Limit 2
//     PlcTask Inputs/GVL_iXlinker.EtherCAT_Master_ELXxxxx.Beckhoff_ELXxxxx.A_0020_ELX3314_0000_0016.TC_Inputs_Channel_1.Status/Error <-> TC Inputs Channel 1/Status/Error
//     PlcTask Inputs/GVL_iXlinker.EtherCAT_Master_ELXxxxx.Beckhoff_ELXxxxx.A_0020_ELX3314_0000_0016.TC_Inputs_Channel_2.Status/Error <-> TC Inputs Channel 2/Status/Error
//     PlcTask Inputs/GVL_iXlinker.EtherCAT_Master_ELXxxxx.Beckhoff_ELXxxxx.A_0020_ELX3314_0000_0016.TC_Inputs_Channel_3.Status/Error <-> TC Inputs Channel 3/Status/Error
//     PlcTask Inputs/GVL_iXlinker.EtherCAT_Master_ELXxxxx.Beckhoff_ELXxxxx.A_0020_ELX3314_0000_0016.TC_Inputs_Channel_4.Status/Error <-> TC Inputs Channel 4/Status/Error
//     PlcTask Inputs/GVL_iXlinker.EtherCAT_Master_ELXxxxx.Beckhoff_ELXxxxx.A_0020_ELX3314_0000_0016.TC_Inputs_Channel_1.Status/TxPDO_State <-> TC Inputs Channel 1/Status/TxPDO State
//     PlcTask Inputs/GVL_iXlinker.EtherCAT_Master_ELXxxxx.Beckhoff_ELXxxxx.A_0020_ELX3314_0000_0016.TC_Inputs_Channel_2.Status/TxPDO_State <-> TC Inputs Channel 2/Status/TxPDO State
//     PlcTask Inputs/GVL_iXlinker.EtherCAT_Master_ELXxxxx.Beckhoff_ELXxxxx.A_0020_ELX3314_0000_0016.TC_Inputs_Channel_3.Status/TxPDO_State <-> TC Inputs Channel 3/Status/TxPDO State
//     PlcTask Inputs/GVL_iXlinker.EtherCAT_Master_ELXxxxx.Beckhoff_ELXxxxx.A_0020_ELX3314_0000_0016.TC_Inputs_Channel_4.Status/TxPDO_State <-> TC Inputs Channel 4/Status/TxPDO State
//     PlcTask Inputs/GVL_iXlinker.EtherCAT_Master_ELXxxxx.Beckhoff_ELXxxxx.A_0020_ELX3314_0000_0016.TC_Inputs_Channel_1.Status/TxPDO_Toggle <-> TC Inputs Channel 1/Status/TxPDO Toggle
//     PlcTask Inputs/GVL_iXlinker.EtherCAT_Master_ELXxxxx.Beckhoff_ELXxxxx.A_0020_ELX3314_0000_0016.TC_Inputs_Channel_2.Status/TxPDO_Toggle <-> TC Inputs Channel 2/Status/TxPDO Toggle
//     PlcTask Inputs/GVL_iXlinker.EtherCAT_Master_ELXxxxx.Beckhoff_ELXxxxx.A_0020_ELX3314_0000_0016.TC_Inputs_Channel_3.Status/TxPDO_Toggle <-> TC Inputs Channel 3/Status/TxPDO Toggle
//     PlcTask Inputs/GVL_iXlinker.EtherCAT_Master_ELXxxxx.Beckhoff_ELXxxxx.A_0020_ELX3314_0000_0016.TC_Inputs_Channel_4.Status/TxPDO_Toggle <-> TC Inputs Channel 4/Status/TxPDO Toggle
//     PlcTask Inputs/GVL_iXlinker.EtherCAT_Master_ELXxxxx.Beckhoff_ELXxxxx.A_0020_ELX3314_0000_0016.TC_Inputs_Channel_1.Value <-> TC Inputs Channel 1/Value
//     PlcTask Inputs/GVL_iXlinker.EtherCAT_Master_ELXxxxx.Beckhoff_ELXxxxx.A_0020_ELX3314_0000_0016.TC_Inputs_Channel_2.Value <-> TC Inputs Channel 2/Value
//     PlcTask Inputs/GVL_iXlinker.EtherCAT_Master_ELXxxxx.Beckhoff_ELXxxxx.A_0020_ELX3314_0000_0016.TC_Inputs_Channel_3.Value <-> TC Inputs Channel 3/Value
//     PlcTask Inputs/GVL_iXlinker.EtherCAT_Master_ELXxxxx.Beckhoff_ELXxxxx.A_0020_ELX3314_0000_0016.TC_Inputs_Channel_4.Value <-> TC Inputs Channel 4/Value
//     PlcTask Inputs/GVL_iXlinker.EtherCAT_Master_ELXxxxx.Beckhoff_ELXxxxx.A_0020_ELX3314_0000_0016.WcState.WcState <-> WcState/WcState
//     PlcTask Inputs/GVL_iXlinker.EtherCAT_Master_ELXxxxx.Beckhoff_ELXxxxx.A_0020_ELX3314_0000_0016.WcState.InputToggle <-> WcState/InputToggle
//     PlcTask Inputs/GVL_iXlinker.EtherCAT_Master_ELXxxxx.Beckhoff_ELXxxxx.A_0020_ELX3314_0000_0016.InfoData.AdsAddr <-> InfoData/AdsAddr
//     PlcTask Inputs/GVL_iXlinker.EtherCAT_Master_ELXxxxx.Beckhoff_ELXxxxx.A_0020_ELX3314_0000_0016.InfoData.State <-> InfoData/State
//   PLC/PLC Instance <-> EtherCAT Master ELXxxxx/Beckhoff ELXxxxx/A_0021(ELX3314-0090-0016)
//     PlcTask Inputs/GVL_iXlinker.EtherCAT_Master_ELXxxxx.Beckhoff_ELXxxxx.A_0021_ELX3314_0090_0016.TC_Inputs_Channel_1.Status/Underrange <-> TC Inputs Channel 1/Status/Underrange
//     PlcTask Inputs/GVL_iXlinker.EtherCAT_Master_ELXxxxx.Beckhoff_ELXxxxx.A_0021_ELX3314_0090_0016.TC_Inputs_Channel_2.Status/Underrange <-> TC Inputs Channel 2/Status/Underrange
//     PlcTask Inputs/GVL_iXlinker.EtherCAT_Master_ELXxxxx.Beckhoff_ELXxxxx.A_0021_ELX3314_0090_0016.TC_Inputs_Channel_3.Status/Underrange <-> TC Inputs Channel 3/Status/Underrange
//     PlcTask Inputs/GVL_iXlinker.EtherCAT_Master_ELXxxxx.Beckhoff_ELXxxxx.A_0021_ELX3314_0090_0016.TC_Inputs_Channel_4.Status/Underrange <-> TC Inputs Channel 4/Status/Underrange
//     PlcTask Inputs/GVL_iXlinker.EtherCAT_Master_ELXxxxx.Beckhoff_ELXxxxx.A_0021_ELX3314_0090_0016.TC_Inputs_Channel_1.Status/Overrange <-> TC Inputs Channel 1/Status/Overrange
//     PlcTask Inputs/GVL_iXlinker.EtherCAT_Master_ELXxxxx.Beckhoff_ELXxxxx.A_0021_ELX3314_0090_0016.TC_Inputs_Channel_2.Status/Overrange <-> TC Inputs Channel 2/Status/Overrange
//     PlcTask Inputs/GVL_iXlinker.EtherCAT_Master_ELXxxxx.Beckhoff_ELXxxxx.A_0021_ELX3314_0090_0016.TC_Inputs_Channel_3.Status/Overrange <-> TC Inputs Channel 3/Status/Overrange
//     PlcTask Inputs/GVL_iXlinker.EtherCAT_Master_ELXxxxx.Beckhoff_ELXxxxx.A_0021_ELX3314_0090_0016.TC_Inputs_Channel_4.Status/Overrange <-> TC Inputs Channel 4/Status/Overrange
//     PlcTask Inputs/GVL_iXlinker.EtherCAT_Master_ELXxxxx.Beckhoff_ELXxxxx.A_0021_ELX3314_0090_0016.TC_Inputs_Channel_1.Status/Limit_1 <-> TC Inputs Channel 1/Status/Limit 1
//     PlcTask Inputs/GVL_iXlinker.EtherCAT_Master_ELXxxxx.Beckhoff_ELXxxxx.A_0021_ELX3314_0090_0016.TC_Inputs_Channel_1.Status/Limit_2 <-> TC Inputs Channel 1/Status/Limit 2
//     PlcTask Inputs/GVL_iXlinker.EtherCAT_Master_ELXxxxx.Beckhoff_ELXxxxx.A_0021_ELX3314_0090_0016.TC_Inputs_Channel_2.Status/Limit_1 <-> TC Inputs Channel 2/Status/Limit 1
//     PlcTask Inputs/GVL_iXlinker.EtherCAT_Master_ELXxxxx.Beckhoff_ELXxxxx.A_0021_ELX3314_0090_0016.TC_Inputs_Channel_2.Status/Limit_2 <-> TC Inputs Channel 2/Status/Limit 2
//     PlcTask Inputs/GVL_iXlinker.EtherCAT_Master_ELXxxxx.Beckhoff_ELXxxxx.A_0021_ELX3314_0090_0016.TC_Inputs_Channel_3.Status/Limit_1 <-> TC Inputs Channel 3/Status/Limit 1
//     PlcTask Inputs/GVL_iXlinker.EtherCAT_Master_ELXxxxx.Beckhoff_ELXxxxx.A_0021_ELX3314_0090_0016.TC_Inputs_Channel_3.Status/Limit_2 <-> TC Inputs Channel 3/Status/Limit 2
//     PlcTask Inputs/GVL_iXlinker.EtherCAT_Master_ELXxxxx.Beckhoff_ELXxxxx.A_0021_ELX3314_0090_0016.TC_Inputs_Channel_4.Status/Limit_1 <-> TC Inputs Channel 4/Status/Limit 1
//     PlcTask Inputs/GVL_iXlinker.EtherCAT_Master_ELXxxxx.Beckhoff_ELXxxxx.A_0021_ELX3314_0090_0016.TC_Inputs_Channel_4.Status/Limit_2 <-> TC Inputs Channel 4/Status/Limit 2
//     PlcTask Inputs/GVL_iXlinker.EtherCAT_Master_ELXxxxx.Beckhoff_ELXxxxx.A_0021_ELX3314_0090_0016.TC_Inputs_Channel_1.Status/Error <-> TC Inputs Channel 1/Status/Error
//     PlcTask Inputs/GVL_iXlinker.EtherCAT_Master_ELXxxxx.Beckhoff_ELXxxxx.A_0021_ELX3314_0090_0016.TC_Inputs_Channel_2.Status/Error <-> TC Inputs Channel 2/Status/Error
//     PlcTask Inputs/GVL_iXlinker.EtherCAT_Master_ELXxxxx.Beckhoff_ELXxxxx.A_0021_ELX3314_0090_0016.TC_Inputs_Channel_3.Status/Error <-> TC Inputs Channel 3/Status/Error
//     PlcTask Inputs/GVL_iXlinker.EtherCAT_Master_ELXxxxx.Beckhoff_ELXxxxx.A_0021_ELX3314_0090_0016.TC_Inputs_Channel_4.Status/Error <-> TC Inputs Channel 4/Status/Error
//     PlcTask Inputs/GVL_iXlinker.EtherCAT_Master_ELXxxxx.Beckhoff_ELXxxxx.A_0021_ELX3314_0090_0016.TC_Inputs_Channel_1.Status/TxPDO_State <-> TC Inputs Channel 1/Status/TxPDO State
//     PlcTask Inputs/GVL_iXlinker.EtherCAT_Master_ELXxxxx.Beckhoff_ELXxxxx.A_0021_ELX3314_0090_0016.TC_Inputs_Channel_2.Status/TxPDO_State <-> TC Inputs Channel 2/Status/TxPDO State
//     PlcTask Inputs/GVL_iXlinker.EtherCAT_Master_ELXxxxx.Beckhoff_ELXxxxx.A_0021_ELX3314_0090_0016.TC_Inputs_Channel_3.Status/TxPDO_State <-> TC Inputs Channel 3/Status/TxPDO State
//     PlcTask Inputs/GVL_iXlinker.EtherCAT_Master_ELXxxxx.Beckhoff_ELXxxxx.A_0021_ELX3314_0090_0016.TC_Inputs_Channel_4.Status/TxPDO_State <-> TC Inputs Channel 4/Status/TxPDO State
//     PlcTask Inputs/GVL_iXlinker.EtherCAT_Master_ELXxxxx.Beckhoff_ELXxxxx.A_0021_ELX3314_0090_0016.TC_Inputs_Channel_1.Status/TxPDO_Toggle <-> TC Inputs Channel 1/Status/TxPDO Toggle
//     PlcTask Inputs/GVL_iXlinker.EtherCAT_Master_ELXxxxx.Beckhoff_ELXxxxx.A_0021_ELX3314_0090_0016.TC_Inputs_Channel_2.Status/TxPDO_Toggle <-> TC Inputs Channel 2/Status/TxPDO Toggle
//     PlcTask Inputs/GVL_iXlinker.EtherCAT_Master_ELXxxxx.Beckhoff_ELXxxxx.A_0021_ELX3314_0090_0016.TC_Inputs_Channel_3.Status/TxPDO_Toggle <-> TC Inputs Channel 3/Status/TxPDO Toggle
//     PlcTask Inputs/GVL_iXlinker.EtherCAT_Master_ELXxxxx.Beckhoff_ELXxxxx.A_0021_ELX3314_0090_0016.TC_Inputs_Channel_4.Status/TxPDO_Toggle <-> TC Inputs Channel 4/Status/TxPDO Toggle
//     PlcTask Inputs/GVL_iXlinker.EtherCAT_Master_ELXxxxx.Beckhoff_ELXxxxx.A_0021_ELX3314_0090_0016.TC_Inputs_Channel_1.Value <-> TC Inputs Channel 1/Value
//     PlcTask Inputs/GVL_iXlinker.EtherCAT_Master_ELXxxxx.Beckhoff_ELXxxxx.A_0021_ELX3314_0090_0016.TC_Inputs_Channel_2.Value <-> TC Inputs Channel 2/Value
//     PlcTask Inputs/GVL_iXlinker.EtherCAT_Master_ELXxxxx.Beckhoff_ELXxxxx.A_0021_ELX3314_0090_0016.TC_Inputs_Channel_3.Value <-> TC Inputs Channel 3/Value
//     PlcTask Inputs/GVL_iXlinker.EtherCAT_Master_ELXxxxx.Beckhoff_ELXxxxx.A_0021_ELX3314_0090_0016.TC_Inputs_Channel_4.Value <-> TC Inputs Channel 4/Value
//     PlcTask Inputs/GVL_iXlinker.EtherCAT_Master_ELXxxxx.Beckhoff_ELXxxxx.A_0021_ELX3314_0090_0016.WcState.WcState <-> WcState/WcState
//     PlcTask Inputs/GVL_iXlinker.EtherCAT_Master_ELXxxxx.Beckhoff_ELXxxxx.A_0021_ELX3314_0090_0016.WcState.InputToggle <-> WcState/InputToggle
//     PlcTask Inputs/GVL_iXlinker.EtherCAT_Master_ELXxxxx.Beckhoff_ELXxxxx.A_0021_ELX3314_0090_0016.InfoData.AdsAddr <-> InfoData/AdsAddr
//     PlcTask Inputs/GVL_iXlinker.EtherCAT_Master_ELXxxxx.Beckhoff_ELXxxxx.A_0021_ELX3314_0090_0016.InfoData.State <-> InfoData/State
//   PLC/PLC Instance <-> EtherCAT Master ELXxxxx/Beckhoff ELXxxxx/A_0022(ELX3351-0000-0016)
//     PlcTask Inputs/GVL_iXlinker.EtherCAT_Master_ELXxxxx.Beckhoff_ELXxxxx.A_0022_ELX3351_0000_0016.RMB_Status.Status/Overrange <-> RMB Status/Status/Overrange
//     PlcTask Inputs/GVL_iXlinker.EtherCAT_Master_ELXxxxx.Beckhoff_ELXxxxx.A_0022_ELX3351_0000_0016.RMB_Status.Status/Data_invalid <-> RMB Status/Status/Data invalid
//     PlcTask Inputs/GVL_iXlinker.EtherCAT_Master_ELXxxxx.Beckhoff_ELXxxxx.A_0022_ELX3351_0000_0016.RMB_Status.Status/Error <-> RMB Status/Status/Error
//     PlcTask Inputs/GVL_iXlinker.EtherCAT_Master_ELXxxxx.Beckhoff_ELXxxxx.A_0022_ELX3351_0000_0016.RMB_Status.Status/Calibration_in_progress <-> RMB Status/Status/Calibration in progress
//     PlcTask Inputs/GVL_iXlinker.EtherCAT_Master_ELXxxxx.Beckhoff_ELXxxxx.A_0022_ELX3351_0000_0016.RMB_Status.Status/Steady_state <-> RMB Status/Status/Steady state
//     PlcTask Inputs/GVL_iXlinker.EtherCAT_Master_ELXxxxx.Beckhoff_ELXxxxx.A_0022_ELX3351_0000_0016.RMB_Status.Status/TxPDO_Toggle <-> RMB Status/Status/TxPDO Toggle
//     PlcTask Inputs/GVL_iXlinker.EtherCAT_Master_ELXxxxx.Beckhoff_ELXxxxx.A_0022_ELX3351_0000_0016.RMB_Value_INT32.Value <-> RMB Value (INT32)/Value
//     PlcTask Outputs/GVL_iXlinker.EtherCAT_Master_ELXxxxx.Beckhoff_ELXxxxx.A_0022_ELX3351_0000_0016.RMB_Control.Ctrl/Start_calibration <-> RMB Control/Ctrl/Start calibration
//     PlcTask Outputs/GVL_iXlinker.EtherCAT_Master_ELXxxxx.Beckhoff_ELXxxxx.A_0022_ELX3351_0000_0016.RMB_Control.Ctrl/Disable_calibration <-> RMB Control/Ctrl/Disable calibration
//     PlcTask Outputs/GVL_iXlinker.EtherCAT_Master_ELXxxxx.Beckhoff_ELXxxxx.A_0022_ELX3351_0000_0016.RMB_Control.Ctrl/Input_freeze <-> RMB Control/Ctrl/Input freeze
//     PlcTask Outputs/GVL_iXlinker.EtherCAT_Master_ELXxxxx.Beckhoff_ELXxxxx.A_0022_ELX3351_0000_0016.RMB_Control.Ctrl/Tara <-> RMB Control/Ctrl/Tara
//     PlcTask Inputs/GVL_iXlinker.EtherCAT_Master_ELXxxxx.Beckhoff_ELXxxxx.A_0022_ELX3351_0000_0016.WcState.WcState <-> WcState/WcState
//     PlcTask Inputs/GVL_iXlinker.EtherCAT_Master_ELXxxxx.Beckhoff_ELXxxxx.A_0022_ELX3351_0000_0016.WcState.InputToggle <-> WcState/InputToggle
//     PlcTask Inputs/GVL_iXlinker.EtherCAT_Master_ELXxxxx.Beckhoff_ELXxxxx.A_0022_ELX3351_0000_0016.InfoData.AdsAddr <-> InfoData/AdsAddr
//     PlcTask Inputs/GVL_iXlinker.EtherCAT_Master_ELXxxxx.Beckhoff_ELXxxxx.A_0022_ELX3351_0000_0016.InfoData.State <-> InfoData/State
//   PLC/PLC Instance <-> EtherCAT Master ELXxxxx/Beckhoff ELXxxxx/A_0023(ELX3351-0090-0016)
//     PlcTask Inputs/GVL_iXlinker.EtherCAT_Master_ELXxxxx.Beckhoff_ELXxxxx.A_0023_ELX3351_0090_0016.RMB_Status.Status/Overrange <-> RMB Status/Status/Overrange
//     PlcTask Inputs/GVL_iXlinker.EtherCAT_Master_ELXxxxx.Beckhoff_ELXxxxx.A_0023_ELX3351_0090_0016.RMB_Status.Status/Data_invalid <-> RMB Status/Status/Data invalid
//     PlcTask Inputs/GVL_iXlinker.EtherCAT_Master_ELXxxxx.Beckhoff_ELXxxxx.A_0023_ELX3351_0090_0016.RMB_Status.Status/Error <-> RMB Status/Status/Error
//     PlcTask Inputs/GVL_iXlinker.EtherCAT_Master_ELXxxxx.Beckhoff_ELXxxxx.A_0023_ELX3351_0090_0016.RMB_Status.Status/Calibration_in_progress <-> RMB Status/Status/Calibration in progress
//     PlcTask Inputs/GVL_iXlinker.EtherCAT_Master_ELXxxxx.Beckhoff_ELXxxxx.A_0023_ELX3351_0090_0016.RMB_Status.Status/Steady_state <-> RMB Status/Status/Steady state
//     PlcTask Inputs/GVL_iXlinker.EtherCAT_Master_ELXxxxx.Beckhoff_ELXxxxx.A_0023_ELX3351_0090_0016.RMB_Status.Status/TxPDO_Toggle <-> RMB Status/Status/TxPDO Toggle
//     PlcTask Inputs/GVL_iXlinker.EtherCAT_Master_ELXxxxx.Beckhoff_ELXxxxx.A_0023_ELX3351_0090_0016.RMB_Value_INT32.Value <-> RMB Value (INT32)/Value
//     PlcTask Outputs/GVL_iXlinker.EtherCAT_Master_ELXxxxx.Beckhoff_ELXxxxx.A_0023_ELX3351_0090_0016.RMB_Control.Ctrl/Start_calibration <-> RMB Control/Ctrl/Start calibration
//     PlcTask Outputs/GVL_iXlinker.EtherCAT_Master_ELXxxxx.Beckhoff_ELXxxxx.A_0023_ELX3351_0090_0016.RMB_Control.Ctrl/Disable_calibration <-> RMB Control/Ctrl/Disable calibration
//     PlcTask Outputs/GVL_iXlinker.EtherCAT_Master_ELXxxxx.Beckhoff_ELXxxxx.A_0023_ELX3351_0090_0016.RMB_Control.Ctrl/Input_freeze <-> RMB Control/Ctrl/Input freeze
//     PlcTask Outputs/GVL_iXlinker.EtherCAT_Master_ELXxxxx.Beckhoff_ELXxxxx.A_0023_ELX3351_0090_0016.RMB_Control.Ctrl/Tara <-> RMB Control/Ctrl/Tara
//     PlcTask Inputs/GVL_iXlinker.EtherCAT_Master_ELXxxxx.Beckhoff_ELXxxxx.A_0023_ELX3351_0090_0016.WcState.WcState <-> WcState/WcState
//     PlcTask Inputs/GVL_iXlinker.EtherCAT_Master_ELXxxxx.Beckhoff_ELXxxxx.A_0023_ELX3351_0090_0016.WcState.InputToggle <-> WcState/InputToggle
//     PlcTask Inputs/GVL_iXlinker.EtherCAT_Master_ELXxxxx.Beckhoff_ELXxxxx.A_0023_ELX3351_0090_0016.InfoData.AdsAddr <-> InfoData/AdsAddr
//     PlcTask Inputs/GVL_iXlinker.EtherCAT_Master_ELXxxxx.Beckhoff_ELXxxxx.A_0023_ELX3351_0090_0016.InfoData.State <-> InfoData/State
//   PLC/PLC Instance <-> EtherCAT Master ELXxxxx/Beckhoff ELXxxxx/A_0024(ELX4154-0000-0016)
//     PlcTask Outputs/GVL_iXlinker.EtherCAT_Master_ELXxxxx.Beckhoff_ELXxxxx.A_0024_ELX4154_0000_0016.AO_Outputs_Channel_1.Analog_output <-> AO Outputs Channel 1/Analog output
//     PlcTask Outputs/GVL_iXlinker.EtherCAT_Master_ELXxxxx.Beckhoff_ELXxxxx.A_0024_ELX4154_0000_0016.AO_Outputs_Channel_2.Analog_output <-> AO Outputs Channel 2/Analog output
//     PlcTask Outputs/GVL_iXlinker.EtherCAT_Master_ELXxxxx.Beckhoff_ELXxxxx.A_0024_ELX4154_0000_0016.AO_Outputs_Channel_3.Analog_output <-> AO Outputs Channel 3/Analog output
//     PlcTask Outputs/GVL_iXlinker.EtherCAT_Master_ELXxxxx.Beckhoff_ELXxxxx.A_0024_ELX4154_0000_0016.AO_Outputs_Channel_4.Analog_output <-> AO Outputs Channel 4/Analog output
//     PlcTask Inputs/GVL_iXlinker.EtherCAT_Master_ELXxxxx.Beckhoff_ELXxxxx.A_0024_ELX4154_0000_0016.WcState.WcState <-> WcState/WcState
//     PlcTask Inputs/GVL_iXlinker.EtherCAT_Master_ELXxxxx.Beckhoff_ELXxxxx.A_0024_ELX4154_0000_0016.InfoData.AdsAddr <-> InfoData/AdsAddr
//     PlcTask Inputs/GVL_iXlinker.EtherCAT_Master_ELXxxxx.Beckhoff_ELXxxxx.A_0024_ELX4154_0000_0016.InfoData.State <-> InfoData/State
//   PLC/PLC Instance <-> EtherCAT Master ELXxxxx/Beckhoff ELXxxxx/A_0025(ELX4181-0000-0016)
//     PlcTask Outputs/GVL_iXlinker.EtherCAT_Master_ELXxxxx.Beckhoff_ELXxxxx.A_0025_ELX4181_0000_0016.Ch_1.AO_Outputs.Analog_output <-> Ch. 1/AO Outputs/Analog output
//     PlcTask Inputs/GVL_iXlinker.EtherCAT_Master_ELXxxxx.Beckhoff_ELXxxxx.A_0025_ELX4181_0000_0016.WcState.WcState <-> WcState/WcState
//     PlcTask Inputs/GVL_iXlinker.EtherCAT_Master_ELXxxxx.Beckhoff_ELXxxxx.A_0025_ELX4181_0000_0016.InfoData.AdsAddr <-> InfoData/AdsAddr
//     PlcTask Inputs/GVL_iXlinker.EtherCAT_Master_ELXxxxx.Beckhoff_ELXxxxx.A_0025_ELX4181_0000_0016.InfoData.AoeNetId <-> InfoData/AoeNetId
//     PlcTask Inputs/GVL_iXlinker.EtherCAT_Master_ELXxxxx.Beckhoff_ELXxxxx.A_0025_ELX4181_0000_0016.InfoData.State <-> InfoData/State
//   PLC/PLC Instance <-> EtherCAT Master ELXxxxx/Beckhoff ELXxxxx/A_0026(ELX4181-0000-0017)
//     PlcTask Outputs/GVL_iXlinker.EtherCAT_Master_ELXxxxx.Beckhoff_ELXxxxx.A_0026_ELX4181_0000_0017.Ch_1.AO_Outputs.Analog_output <-> Ch. 1/AO Outputs/Analog output
//     PlcTask Inputs/GVL_iXlinker.EtherCAT_Master_ELXxxxx.Beckhoff_ELXxxxx.A_0026_ELX4181_0000_0017.WcState.WcState <-> WcState/WcState
//     PlcTask Inputs/GVL_iXlinker.EtherCAT_Master_ELXxxxx.Beckhoff_ELXxxxx.A_0026_ELX4181_0000_0017.InfoData.AdsAddr <-> InfoData/AdsAddr
//     PlcTask Inputs/GVL_iXlinker.EtherCAT_Master_ELXxxxx.Beckhoff_ELXxxxx.A_0026_ELX4181_0000_0017.InfoData.AoeNetId <-> InfoData/AoeNetId
//     PlcTask Inputs/GVL_iXlinker.EtherCAT_Master_ELXxxxx.Beckhoff_ELXxxxx.A_0026_ELX4181_0000_0017.InfoData.State <-> InfoData/State
//   PLC/PLC Instance <-> EtherCAT Master ELXxxxx/Beckhoff ELXxxxx/A_0027(ELX5151-0000-0016)
//     PlcTask Inputs/GVL_iXlinker.EtherCAT_Master_ELXxxxx.Beckhoff_ELXxxxx.A_0027_ELX5151_0000_0016.ENC_Status_compact.Status/Set_counter_done <-> ENC Status compact/Status/Set counter done
//     PlcTask Inputs/GVL_iXlinker.EtherCAT_Master_ELXxxxx.Beckhoff_ELXxxxx.A_0027_ELX5151_0000_0016.ENC_Status_compact.Status/Open_circuit <-> ENC Status compact/Status/Open circuit
//     PlcTask Inputs/GVL_iXlinker.EtherCAT_Master_ELXxxxx.Beckhoff_ELXxxxx.A_0027_ELX5151_0000_0016.ENC_Status_compact.Status/Extrapolation_stall <-> ENC Status compact/Status/Extrapolation stall
//     PlcTask Inputs/GVL_iXlinker.EtherCAT_Master_ELXxxxx.Beckhoff_ELXxxxx.A_0027_ELX5151_0000_0016.ENC_Status_compact.Status/Status_of_input_A <-> ENC Status compact/Status/Status of input A
//     PlcTask Inputs/GVL_iXlinker.EtherCAT_Master_ELXxxxx.Beckhoff_ELXxxxx.A_0027_ELX5151_0000_0016.ENC_Status_compact.Status/Status_of_input_B <-> ENC Status compact/Status/Status of input B
//     PlcTask Inputs/GVL_iXlinker.EtherCAT_Master_ELXxxxx.Beckhoff_ELXxxxx.A_0027_ELX5151_0000_0016.ENC_Status_compact.Status/Sync_error <-> ENC Status compact/Status/Sync error
